REGION Network 9: Clear IDs from HMI if not on that screen
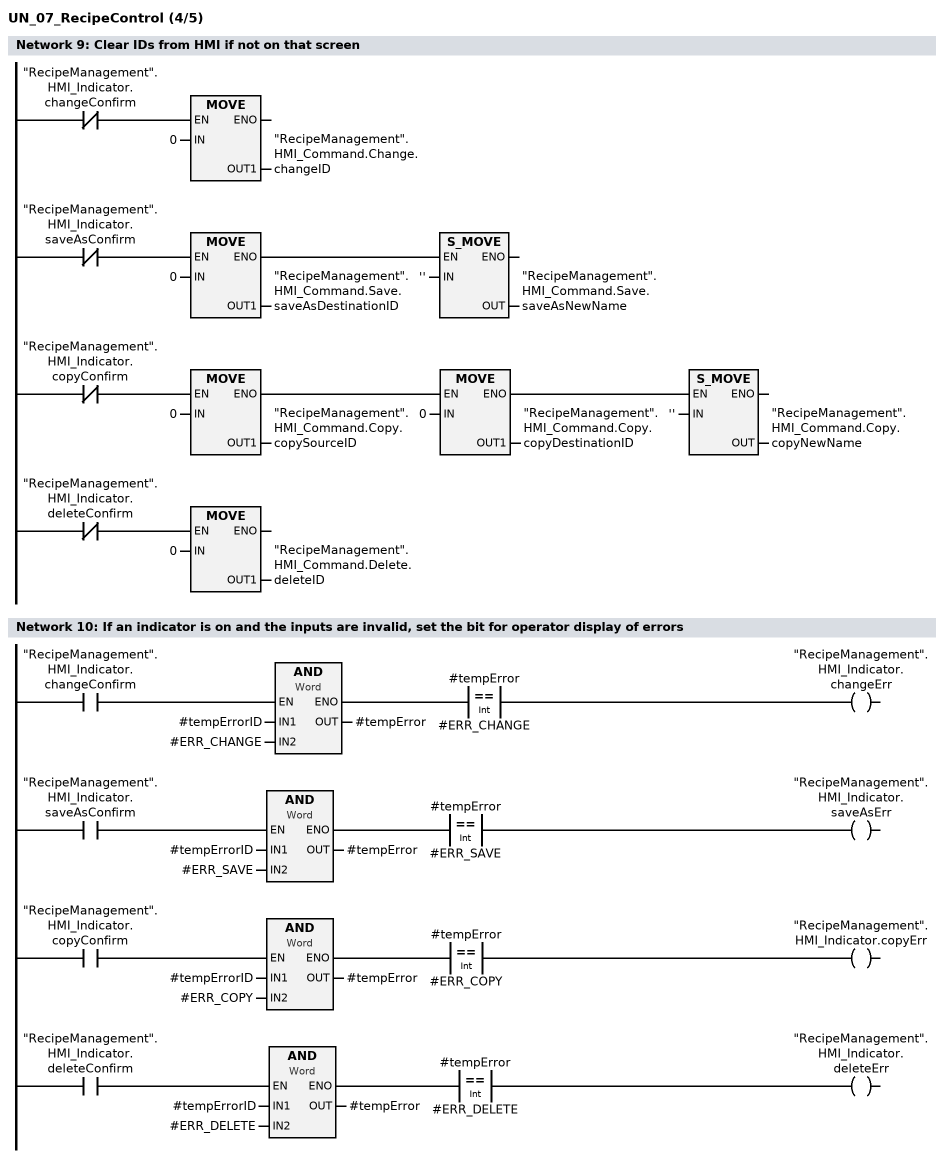
   RUNG wire#powerrail
      I_Contact( "RecipeManagement".HMI_Indicator.changeConfirm )
      Move(in := 0, out1 => "RecipeManagement".HMI_Command.Change.changeID)
   END_RUNG
   RUNG wire#powerrail
      I_Contact( "RecipeManagement".HMI_Indicator.saveAsConfirm )
      Move(in := 0, out1 => "RecipeManagement".HMI_Command.Save.saveAsDestinationID)
      S_Move(in := '', out => "RecipeManagement".HMI_Command.Save.saveAsNewName)
   END_RUNG
   RUNG wire#powerrail
      I_Contact( "RecipeManagement".HMI_Indicator.copyConfirm )
      Move(in := 0, out1 => "RecipeManagement".HMI_Command.Copy.copySourceID)
      Move(in := 0, out1 => "RecipeManagement".HMI_Command.Copy.copyDestinationID)
      S_Move(in := '', out => "RecipeManagement".HMI_Command.Copy.copyNewName)
   END_RUNG
   RUNG wire#powerrail
      I_Contact( "RecipeManagement".HMI_Indicator.deleteConfirm )
      Move(in := 0, out1 => "RecipeManagement".HMI_Command.Delete.deleteID)
   END_RUNG
   // the same network as SCL:
   IF NOT "RecipeManagement".HMI_Indicator.changeConfirm THEN
       "RecipeManagement".HMI_Command.Change.changeID := 0;
   END_IF;
   IF NOT "RecipeManagement".HMI_Indicator.saveAsConfirm THEN
       "RecipeManagement".HMI_Command.Save.saveAsDestinationID := 0;
       "RecipeManagement".HMI_Command.Save.saveAsNewName := '';
   END_IF;
   IF NOT "RecipeManagement".HMI_Indicator.copyConfirm THEN
       "RecipeManagement".HMI_Command.Copy.copySourceID := 0;
       "RecipeManagement".HMI_Command.Copy.copyDestinationID := 0;
       "RecipeManagement".HMI_Command.Copy.copyNewName := '';
   END_IF;
   IF NOT "RecipeManagement".HMI_Indicator.deleteConfirm THEN
       "RecipeManagement".HMI_Command.Delete.deleteID := 0;
   END_IF;
END_REGION

REGION Network 10: If an indicator is on and the inputs are invalid, set the bit for operator display of errors
   RUNG wire#powerrail
      Contact( "RecipeManagement".HMI_Indicator.changeConfirm )
      { S7_Templates := "SrcType := Word" } And(in1 := #tempErrorID, in2 := #ERR_CHANGE, out => #tempError)
      { S7_Templates := "SrcType := Int" } EQ_Contact(in1 := #tempError, in2 := #ERR_CHANGE)
      Coil( "RecipeManagement".HMI_Indicator.changeErr )
   END_RUNG
   RUNG wire#powerrail
      Contact( "RecipeManagement".HMI_Indicator.saveAsConfirm )
      { S7_Templates := "SrcType := Word" } And(in1 := #tempErrorID, in2 := #ERR_SAVE, out => #tempError)
      { S7_Templates := "SrcType := Int" } EQ_Contact(in1 := #tempError, in2 := #ERR_SAVE)
      Coil( "RecipeManagement".HMI_Indicator.saveAsErr )
   END_RUNG
   RUNG wire#powerrail
      Contact( "RecipeManagement".HMI_Indicator.copyConfirm )
      { S7_Templates := "SrcType := Word" } And(in1 := #tempErrorID, in2 := #ERR_COPY, out => #tempError)
      { S7_Templates := "SrcType := Int" } EQ_Contact(in1 := #tempError, in2 := #ERR_COPY)
      Coil( "RecipeManagement".HMI_Indicator.copyErr )
   END_RUNG
   RUNG wire#powerrail
      Contact( "RecipeManagement".HMI_Indicator.deleteConfirm )
      { S7_Templates := "SrcType := Word" } And(in1 := #tempErrorID, in2 := #ERR_DELETE, out => #tempError)
      { S7_Templates := "SrcType := Int" } EQ_Contact(in1 := #tempError, in2 := #ERR_DELETE)
      Coil( "RecipeManagement".HMI_Indicator.deleteErr )
   END_RUNG
   // the same network as SCL:
   IF "RecipeManagement".HMI_Indicator.changeConfirm THEN #tempError := #tempErrorID AND #ERR_CHANGE; END_IF;
   "RecipeManagement".HMI_Indicator.changeErr := "RecipeManagement".HMI_Indicator.changeConfirm AND (#tempError = #ERR_CHANGE);
   IF "RecipeManagement".HMI_Indicator.saveAsConfirm THEN #tempError := #tempErrorID AND #ERR_SAVE; END_IF;
   "RecipeManagement".HMI_Indicator.saveAsErr := "RecipeManagement".HMI_Indicator.saveAsConfirm AND (#tempError = #ERR_SAVE);
   IF "RecipeManagement".HMI_Indicator.copyConfirm THEN #tempError := #tempErrorID AND #ERR_COPY; END_IF;
   "RecipeManagement".HMI_Indicator.copyErr := "RecipeManagement".HMI_Indicator.copyConfirm AND (#tempError = #ERR_COPY);
   IF "RecipeManagement".HMI_Indicator.deleteConfirm THEN #tempError := #tempErrorID AND #ERR_DELETE; END_IF;
   "RecipeManagement".HMI_Indicator.deleteErr := "RecipeManagement".HMI_Indicator.deleteConfirm AND (#tempError = #ERR_DELETE);
END_REGION

REGION Network 11: Call Recipe HMI Manager to handle display of setpoints
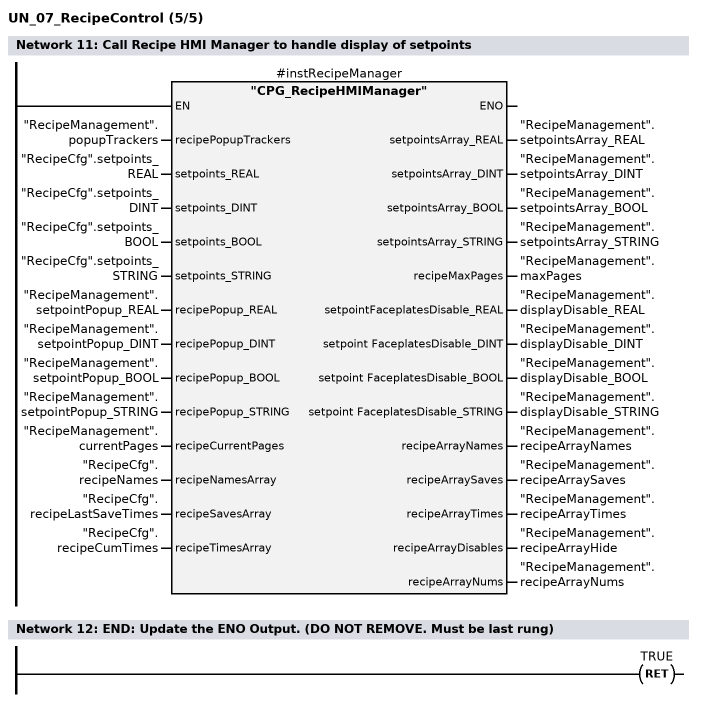
   RUNG wire#powerrail
      #instRecipeManager(recipePopupTrackers := "RecipeManagement".popupTrackers, setpoints_REAL := "RecipeCfg".setpoints_REAL, setpoints_DINT := "RecipeCfg".setpoints_DINT, setpoints_BOOL := "RecipeCfg".setpoints_BOOL, setpoints_STRING := "RecipeCfg".setpoints_STRING, recipePopup_REAL := "RecipeManagement".setpointPopup_REAL, recipePopup_DINT := "RecipeManagement".setpointPopup_DINT, recipePopup_BOOL := "RecipeManagement".setpointPopup_BOOL, recipePopup_STRING := "RecipeManagement".setpointPopup_STRING, recipeCurrentPages := "RecipeManagement".currentPages, recipeNamesArray := "RecipeCfg".recipeNames, recipeSavesArray := "RecipeCfg".recipeLastSaveTimes, recipeTimesArray := "RecipeCfg".recipeCumTimes, setpointsArray_REAL => "RecipeManagement".setpointsArray_REAL, setpointsArray_DINT => "RecipeManagement".setpointsArray_DINT, setpointsArray_BOOL => "RecipeManagement".setpointsArray_BOOL, setpointsArray_STRING => "RecipeManagement".setpointsArray_STRING, recipeMaxPages => "RecipeManagement".maxPages, setpointFaceplatesDisable_REAL => "RecipeManagement".displayDisable_REAL, "setpoint FaceplatesDisable_DINT" => "RecipeManagement".displayDisable_DINT, "setpoint FaceplatesDisable_BOOL" => "RecipeManagement".displayDisable_BOOL, "setpoint FaceplatesDisable_STRING" => "RecipeManagement".displayDisable_STRING, recipeArrayNames => "RecipeManagement".recipeArrayNames, recipeArraySaves => "RecipeManagement".recipeArraySaves, recipeArrayTimes => "RecipeManagement".recipeArrayTimes, recipeArrayDisables => "RecipeManagement".recipeArrayHide, recipeArrayNums => "RecipeManagement".recipeArrayNums)
   END_RUNG
   // the same network as SCL:
   #instRecipeManager(recipePopupTrackers := "RecipeManagement".popupTrackers,   // "CPG_RecipeHMIManager"
                      setpoints_REAL := "RecipeCfg".setpoints_REAL,
                      setpoints_DINT := "RecipeCfg".setpoints_DINT,
                      setpoints_BOOL := "RecipeCfg".setpoints_BOOL,
                      setpoints_STRING := "RecipeCfg".setpoints_STRING,
                      recipePopup_REAL := "RecipeManagement".setpointPopup_REAL,
                      recipePopup_DINT := "RecipeManagement".setpointPopup_DINT,
                      recipePopup_BOOL := "RecipeManagement".setpointPopup_BOOL,
                      recipePopup_STRING := "RecipeManagement".setpointPopup_STRING,
                      recipeCurrentPages := "RecipeManagement".currentPages,
                      recipeNamesArray := "RecipeCfg".recipeNames,
                      recipeSavesArray := "RecipeCfg".recipeLastSaveTimes,
                      recipeTimesArray := "RecipeCfg".recipeCumTimes,
                      setpointsArray_REAL => "RecipeManagement".setpointsArray_REAL,
                      setpointsArray_DINT => "RecipeManagement".setpointsArray_DINT,
                      setpointsArray_BOOL => "RecipeManagement".setpointsArray_BOOL,
                      setpointsArray_STRING => "RecipeManagement".setpointsArray_STRING,
                      recipeMaxPages => "RecipeManagement".maxPages,
                      setpointFaceplatesDisable_REAL => "RecipeManagement".displayDisable_REAL,
                      "setpoint FaceplatesDisable_DINT" => "RecipeManagement".displayDisable_DINT,
                      "setpoint FaceplatesDisable_BOOL" => "RecipeManagement".displayDisable_BOOL,
                      "setpoint FaceplatesDisable_STRING" => "RecipeManagement".displayDisable_STRING,
                      recipeArrayNames => "RecipeManagement".recipeArrayNames,
                      recipeArraySaves => "RecipeManagement".recipeArraySaves,
                      recipeArrayTimes => "RecipeManagement".recipeArrayTimes,
                      recipeArrayDisables => "RecipeManagement".recipeArrayHide,
                      recipeArrayNums => "RecipeManagement".recipeArrayNums);
END_REGION

REGION Network 12: END: Update the ENO Output. (DO NOT REMOVE. Must be last rung)
   RUNG wire#powerrail
      ReturnCoil( TRUE )
   END_RUNG
   // the same network as SCL:
   ENO := TRUE;
   RETURN;
END_REGION
END_FUNCTION_BLOCK

FUNCTION_BLOCK "CPG_RecipeControl"
TITLE = CPG_RecipeControl
{ S7_Optimized_Access := 'TRUE' }
AUTHOR : 'tech.team.motioncontrol@siemens.com'
FAMILY : CPG
VERSION : 1.1
//Support: tech.team.motioncontrol@siemens.com
   VAR_INPUT 
      enable { ExternalAccessible := 'False'; ExternalVisible := 'False'; ExternalWritable := 'False'} : Bool;   // Recipe change is only possible if instruction is enabled
      recipeChangeID { ExternalAccessible := 'False'; ExternalVisible := 'False'; ExternalWritable := 'False'} : Int;   // ID of recipe to change to
      recipeChangeReq { ExternalAccessible := 'False'; ExternalVisible := 'False'; ExternalWritable := 'False'} : Bool;   // Change recipe on rising edge
      recipeSaveReq { ExternalAccessible := 'False'; ExternalVisible := 'False'; ExternalWritable := 'False'} : Bool;   // Save current recipe on rising edge
      recipeSaveAsID { ExternalAccessible := 'False'; ExternalVisible := 'False'; ExternalWritable := 'False'} : Int;   // Location to saveas recipe to
      recipeSaveAsReq { ExternalAccessible := 'False'; ExternalVisible := 'False'; ExternalWritable := 'False'} : Bool;   // SaveAs recipe on rising edge
      recipeCopySourceID { ExternalAccessible := 'False'; ExternalVisible := 'False'; ExternalWritable := 'False'} : Int;   // Location to copy recipe from
      recipeCopyID { ExternalAccessible := 'False'; ExternalVisible := 'False'; ExternalWritable := 'False'} : Int;   // Location to copy recipe to
      recipeCopyReq { ExternalAccessible := 'False'; ExternalVisible := 'False'; ExternalWritable := 'False'} : Bool;   // Copy recipe on rising edge
      newRecipeName { ExternalAccessible := 'False'; ExternalVisible := 'False'; ExternalWritable := 'False'} : String[60];   // Name of the saveas or copied recipe
      recipeDeleteID { ExternalAccessible := 'False'; ExternalVisible := 'False'; ExternalWritable := 'False'} : Int;   // Location of recipe to delete
      recipeDeleteReq { ExternalAccessible := 'False'; ExternalVisible := 'False'; ExternalWritable := 'False'} : Bool;   // Delete recipe on rising edge
      resetAllTimes { ExternalAccessible := 'False'; ExternalVisible := 'False'; ExternalWritable := 'False'} : Bool;   // Reset cumulative seconds for all recipes
   END_VAR

   VAR_OUTPUT 
      currentRecipeID { ExternalAccessible := 'False'; ExternalVisible := 'False'; ExternalWritable := 'False'} : Int;   // ID of the current recipe
      currentRecipeName { ExternalAccessible := 'False'; ExternalVisible := 'False'; ExternalWritable := 'False'} : String[60];   // Name of the current recipe
      recipeChangeDisabled { ExternalAccessible := 'False'; ExternalVisible := 'False'; ExternalWritable := 'False'} : Bool;   // Recipe changes are enabled
      recipeSetpointDiff { ExternalAccessible := 'False'; ExternalVisible := 'False'; ExternalWritable := 'False'} : Bool;   // New setpoint differs from current recipe value
      recipeCurrentSeconds { ExternalAccessible := 'False'; ExternalVisible := 'False'; ExternalWritable := 'False'} : Time;   // Current recipe time in seconds
      error { ExternalAccessible := 'False'; ExternalVisible := 'False'; ExternalWritable := 'False'} : Bool;   // Error Present
      errorID { ExternalAccessible := 'False'; ExternalVisible := 'False'; ExternalWritable := 'False'} : Word := 16#0000;   // Code for Status
   END_VAR

   VAR_IN_OUT 
      recipeControl : "CPG_typeRecipeControl";   // Recipe Control tag
      recipeNames : Array[0.."CPG_NO_OF_RECIPE_UPPER_LIM"] of String[60];   // All recipe names
      recipeCumSeconds : Array[0.."CPG_NO_OF_RECIPE_UPPER_LIM"] of Time;   // Cumulative times for all recipes
      recipeSaveDates {InstructionName := 'DTL'; LibVersion := '1.0'} : Array[0.."CPG_NO_OF_RECIPE_UPPER_LIM"] of DTL;   // Recipe saved date time
   END_VAR

   VAR 
      statSetpoinDiffTimer {InstructionName := 'TON_TIME'; LibVersion := '1.0'; ExternalAccessible := 'False'; ExternalVisible := 'False'; ExternalWritable := 'False'} : TON_TIME;
      statPrevRecipe { ExternalAccessible := 'False'; ExternalVisible := 'False'; ExternalWritable := 'False'} : Int;
      statChangeReq {InstructionName := 'R_TRIG'; LibVersion := '1.0'; ExternalAccessible := 'False'; ExternalVisible := 'False'; ExternalWritable := 'False'} : R_TRIG;
      statSaveReq {InstructionName := 'R_TRIG'; LibVersion := '1.0'; ExternalAccessible := 'False'; ExternalVisible := 'False'; ExternalWritable := 'False'} : R_TRIG;
      statSaveAsReq {InstructionName := 'R_TRIG'; LibVersion := '1.0'; ExternalAccessible := 'False'; ExternalVisible := 'False'; ExternalWritable := 'False'} : R_TRIG;
      statCopyReq {InstructionName := 'R_TRIG'; LibVersion := '1.0'; ExternalAccessible := 'False'; ExternalVisible := 'False'; ExternalWritable := 'False'} : R_TRIG;
      statDeleteReq {InstructionName := 'R_TRIG'; LibVersion := '1.0'; ExternalAccessible := 'False'; ExternalVisible := 'False'; ExternalWritable := 'False'} : R_TRIG;
      statChangeTimer {InstructionName := 'TP_TIME'; LibVersion := '1.0'; ExternalAccessible := 'False'; ExternalVisible := 'False'; ExternalWritable := 'False'} : TP_TIME;
      statChangeTimerFall {InstructionName := 'F_TRIG'; LibVersion := '1.0'; ExternalAccessible := 'False'; ExternalVisible := 'False'; ExternalWritable := 'False'} : F_TRIG;
      statSaveTimer {InstructionName := 'TP_TIME'; LibVersion := '1.0'; ExternalAccessible := 'False'; ExternalVisible := 'False'; ExternalWritable := 'False'} : TP_TIME;
      statSaveTimerFall {InstructionName := 'F_TRIG'; LibVersion := '1.0'; ExternalAccessible := 'False'; ExternalVisible := 'False'; ExternalWritable := 'False'} : F_TRIG;
      statSaveAsTimer {InstructionName := 'TP_TIME'; LibVersion := '1.0'; ExternalAccessible := 'False'; ExternalVisible := 'False'; ExternalWritable := 'False'} : TP_TIME;
      statSaveAsTimerFall {InstructionName := 'F_TRIG'; LibVersion := '1.0'; ExternalAccessible := 'False'; ExternalVisible := 'False'; ExternalWritable := 'False'} : F_TRIG;
      statCopyTimer {InstructionName := 'TP_TIME'; LibVersion := '1.0'; ExternalAccessible := 'False'; ExternalVisible := 'False'; ExternalWritable := 'False'} : TP_TIME;
      statCopyTimerFall {InstructionName := 'F_TRIG'; LibVersion := '1.0'; ExternalAccessible := 'False'; ExternalVisible := 'False'; ExternalWritable := 'False'} : F_TRIG;
      statDeleteTimer {InstructionName := 'TP_TIME'; LibVersion := '1.0'; ExternalAccessible := 'False'; ExternalVisible := 'False'; ExternalWritable := 'False'} : TP_TIME;
      statDeleteTimerFall {InstructionName := 'F_TRIG'; LibVersion := '1.0'; ExternalAccessible := 'False'; ExternalVisible := 'False'; ExternalWritable := 'False'} : F_TRIG;
      statPrevCumSeconds { ExternalAccessible := 'False'; ExternalVisible := 'False'; ExternalWritable := 'False'} : Array[0.."CPG_NO_OF_RECIPE_UPPER_LIM"] of Time;
      statChangeTimeStamp {InstructionName := 'DTL'; LibVersion := '1.0'; ExternalAccessible := 'False'; ExternalVisible := 'False'; ExternalWritable := 'False'} : DTL;
   END_VAR

   VAR_TEMP 
      tempChangeEN : Bool;
      tempCopyRecipeEN : Bool;
      tempSaveRecipeEN : Bool;
      tempDeleteRecipeEN : Bool;
      tempDTLError : Int;
      tempLoop : Int;
      tempTime {InstructionName := 'DTL'; LibVersion := '1.0'} : DTL;
      tempRecipeSaveAs : Bool;
   END_VAR

   VAR CONSTANT 
      MAX_RECIPE_NUM : Int := 20;
      WARNING_TIMERLEN : Time := T#1s;
      CHG_ERR : Word := 16#8001;
      SAVE_ERR : Word := 16#8002;
      COPY_ERR : Word := 16#8004;
      DEL_ERR : Word := 16#8008;
   END_VAR


BEGIN
	//============================================================================================================
	// SIEMENS AG
	// (c)Copyright 2019 All Rights Reserved
	//------------------------------------------------------------------------------------------------------------
	// Library: LCPG
	// Tested with: S7-1500 with FW version V2.1
	// Engineering: TIA Portal V14
	// Restrictions: ---
	// Requirements: S7-1500
	// Functionality: used to control the current machine recipe
	// Support: tech.team.motioncontrol@siemens.com
	//------------------------------------------------------------------------------------------------------------
	// Change log table:
	// Version       Date               Expert in charge    Changes applied
	//  01.01.00     02.01.2019         KB                  Initial Release
	//============================================================================================================
	// Function : CPG_RecipeControl
	//============================================================================================================
	
	REGION INITIALIZATION
	    #errorID := 16#0000;
	    
	    #recipeControl.RecipeChangeDisabled := NOT #enable;
	    
	    //check lanugage for out of bounds
	    IF (#recipeControl.LanguageSelection < 0) OR (#recipeControl.LanguageSelection > "LPMLV30_LANGUAGES_UPPER_LIM") THEN
	        #errorID := #errorID OR 16#1000;
	        #recipeControl.LanguageSelection := 0;
	    END_IF;
	    
	    
	    //Dectect any recipe & setpoint differences
	    //if any call of recipe setpoint FBs has a difference, the RecipeSetpointDiff bit is set
	    IF #recipeControl.RecipeSetpointDiff THEN
	        #recipeSetpointDiff := true;
	        #recipeControl.RecipeSetpointDiff := false;
	    END_IF;
	END_REGION
	
	
	REGION RECIPE MANAGEMENT ENABLING
	    //Check that only 1 recipe command is active
	    IF NOT (#recipeControl.RecipeCopy OR #recipeControl.RecipeDelete OR #recipeControl.RecipeSave) THEN     //all false except change
	        #tempChangeEN := true;
	    END_IF;
	    IF NOT (#recipeControl.RecipeCopy OR #recipeControl.RecipeDelete OR #recipeControl.RecipeChange) THEN   //all false except save/saveas
	        #tempSaveRecipeEN := true;
	    END_IF;
	    IF NOT (#recipeControl.RecipeChange OR #recipeControl.RecipeDelete OR #recipeControl.RecipeSave) THEN   //all false except copy
	        #tempCopyRecipeEN := true;
	    END_IF;
	    IF NOT (#recipeControl.RecipeCopy OR #recipeControl.RecipeChange OR #recipeControl.RecipeSave) THEN     //all false except delete
	        #tempDeleteRecipeEN := true;
	    END_IF;
	    
	    
	    //RecipeCmd out of bounds, or equal to the current recipe
	    IF (#recipeChangeID > #MAX_RECIPE_NUM) OR (#recipeChangeID < 0) OR (#recipeChangeID = #recipeControl.CurrentRecipeID) THEN
	        #errorID := #errorID OR #CHG_ERR;
	        #tempChangeEN := false;
	    END_IF;
	    //RecipeSaveAsCmd out of bounds, or attempting to over current recipe
	    IF (#recipeSaveAsID > #MAX_RECIPE_NUM) OR (#recipeSaveAsID < 0) OR (#recipeSaveAsID = #recipeControl.CurrentRecipeID) THEN
	        #errorID := #errorID OR #SAVE_ERR;
	        #tempSaveRecipeEN := false;
	    END_IF;
	    //RecipeCopyCmd or RecipeCopySourceCmd out of bounds, cannot copy to currently running recipe
	    IF (#recipeCopyID > #MAX_RECIPE_NUM) OR (#recipeCopyID < 0) OR (#recipeCopySourceID > #MAX_RECIPE_NUM) OR (#recipeCopySourceID < 0)
	        OR #recipeCopyID = #recipeControl.CurrentRecipeID THEN
	        #errorID := #errorID OR #COPY_ERR;
	        #tempCopyRecipeEN := false;
	    END_IF;
	    //RecipeDeleteCmd out of bounds or equal to current recipe
	    IF (#recipeDeleteID > #MAX_RECIPE_NUM) OR (#recipeDeleteID < 0) OR (#recipeDeleteID = #recipeControl.CurrentRecipeID) THEN
	        #errorID := #errorID OR #DEL_ERR;
	        #tempDeleteRecipeEN := false;
	    END_IF;
	END_REGION
	
	
	REGION RECIPE CHANGE
	    //only allow recipe changes while enabled
	    IF #enable THEN
	        
	        //timer needed for display & troubleshooting
	        //timer starts on rising edge of the req signal and persists for 1s
	        #statChangeReq(CLK := #recipeChangeReq);
	        
	        #statChangeTimer(IN := #statChangeReq.Q,
	                     PT := #WARNING_TIMERLEN);
	        
	        #statChangeTimerFall(CLK := #statChangeTimer.Q);
	        
	        
	        //Check that the recipe to change is valid & no other command is active
	        IF #tempChangeEN THEN
	            
	            //set output to indicate that a recipe is being changed
	            IF #statChangeTimer.Q THEN
	                #recipeControl.RecipeChange := true;
	            ELSE
	                #recipeControl.RecipeChange := false;
	            END_IF;
	            
	            //change recipe on done bit, true for only 1 scan
	            IF #statChangeTimerFall.Q THEN
	                #recipeControl.RecipeChangeNum := #recipeControl.RecipeChangeNum + 1;
	                #recipeControl.CurrentRecipeID := #recipeChangeID;
	                #recipeControl.CurrentRecipeName := #recipeNames[#recipeControl.CurrentRecipeID];
	            END_IF;
	            
	        END_IF;
	        
	    END_IF;
	END_REGION
	
	
	REGION RECIPE SAVEAS
	    //timer needed for display & troubleshooting
	    //timer starts on rising edge of the req signal and persists for 1s
	    #statSaveAsReq(CLK := #recipeSaveAsReq);
	    
	    #statSaveAsTimer(IN := #statSaveAsReq.Q,
	                 PT := #WARNING_TIMERLEN);
	    
	    #statSaveAsTimerFall(CLK := #statSaveAsTimer.Q);
	    
	    
	    //Check that the recipe to save is valid & no other command is active
	    IF #tempSaveRecipeEN THEN
	        
	        //set output to indicate that a recipe is being saved
	        //because Save & SaveAs use the same output (RecipeControl.RecipeSave), this is handled slightly differently
	        IF #statSaveAsTimer.Q THEN
	            #tempRecipeSaveAs := true;
	        END_IF;
	        
	        
	        //set work variables so that setpoints know the source/destination of the copy operation
	        IF #statSaveAsTimer.Q THEN
	            #recipeControl.RecipeSourceID := #recipeControl.CurrentRecipeID;
	            #recipeControl.RecipeDestinationID := #recipeSaveAsID;
	        END_IF;
	        
	        //update counter, take timestamp, and update recipe name
	        IF #statSaveAsTimerFall.Q THEN
	            #recipeControl.RecipeSaveNum := #recipeControl.RecipeSaveNum + 1;
	            #tempDTLError := RD_LOC_T(#recipeSaveDates[#recipeControl.RecipeDestinationID]);
	            #recipeNames[#recipeControl.RecipeDestinationID] := #newRecipeName;
	        END_IF;
	        
	    END_IF;
	END_REGION
	
	
	REGION RECIPE SAVE
	    //timer needed for display & troubleshooting
	    //timer starts on rising edge of the req signal and persists for 1s
	    #statSaveReq(CLK := #recipeSaveReq);
	    
	    #statSaveTimer(IN := #statSaveReq.Q,
	               PT := #WARNING_TIMERLEN);
	    
	    #statSaveTimerFall(CLK := #statSaveTimer.Q);
	    
	    
	    //saving is always possible
	    //note that the saveas REGION must be after the save REGION
	    //otherwise RecipeControl.RecipeSave won't be set by a saveas
	    
	    //set output to indicate that a recipe is being saved
	    //because Save & SaveAs use the same output (RecipeControl.RecipeSave), this is handled slightly differently
	    IF #statSaveTimer.Q  OR #tempRecipeSaveAs THEN
	        #recipeControl.RecipeSave := true;
	    ELSE
	        #recipeControl.RecipeSave := false;
	    END_IF;
	    
	    //set work variables so that setpoints know the source/destination of the save operation
	    IF #statSaveTimer.Q THEN
	        #recipeControl.RecipeSourceID := #recipeControl.CurrentRecipeID;
	        #recipeControl.RecipeDestinationID := #recipeControl.CurrentRecipeID;
	    END_IF;
	    
	    //update counter, take timestamp
	    IF #statSaveTimerFall.Q THEN
	        #recipeControl.RecipeSaveNum := #recipeControl.RecipeSaveNum + 1;
	        #tempDTLError := RD_LOC_T(#recipeSaveDates[#recipeControl.RecipeDestinationID]);
	    END_IF;
	END_REGION
	
	
	REGION RECIPE COPY
	    //timer needed for display & troubleshooting
	    //timer starts on rising edge of the req signal and persists for 1s
	    #statCopyReq(CLK := #recipeCopyReq);
	    
	    #statCopyTimer(IN := #statCopyReq.Q,
	               PT := #WARNING_TIMERLEN);
	    
	    #statCopyTimerFall(CLK := #statCopyTimer.Q);
	    
	    
	    //Check that the recipes to copy are valid & no other command is active
	    IF #tempCopyRecipeEN THEN
	        
	        //set output to indicate that a recipe is being copied
	        IF #statCopyTimer.Q THEN
	            #recipeControl.RecipeCopy := true;
	        ELSE
	            #recipeControl.RecipeCopy := false;
	        END_IF;
	        
	        //set work variables so that setpoints know the source/destination of the copy operation
	        IF #statCopyTimer.Q THEN
	            #recipeControl.RecipeSourceID := #recipeCopySourceID;
	            #recipeControl.RecipeDestinationID := #recipeCopyID;
	        END_IF;
	        
	        //update the recipename of the new recipe, increment change work variable
	        IF #statCopyTimerFall.Q THEN
	            #recipeControl.RecipeCopyNum := #recipeControl.RecipeCopyNum + 1;
	            #tempDTLError := RD_LOC_T(#recipeSaveDates[#recipeControl.RecipeDestinationID]);
	            #recipeNames[#recipeControl.RecipeDestinationID] := #newRecipeName;
	        END_IF;
	        
	    END_IF;
	END_REGION
	
	
	REGION RECIPE DELETE
	    //timer needed for display & troubleshooting
	    //timer starts on rising edge of the req signal and persists for 1s
	    #statDeleteReq(CLK := #recipeDeleteReq);
	    
	    #statDeleteTimer(IN := #statDeleteReq.Q,
	                 PT := #WARNING_TIMERLEN);
	    
	    #statDeleteTimerFall(CLK := #statDeleteTimer.Q);
	    
	    
	    //Check that the recipe to delete is valid & no other command is active
	    IF #tempDeleteRecipeEN THEN
	        
	        //set output to indicate that a recipe is being copied
	        IF #statDeleteTimer.Q THEN
	            #recipeControl.RecipeDelete := true;
	        ELSE
	            #recipeControl.RecipeDelete := false;
	        END_IF;
	        
	        //set work variable so that setpoints know the destination of the delete operation
	        IF #statDeleteTimer.Q THEN
	            #recipeControl.RecipeDestinationID := #recipeDeleteID;
	        END_IF;
	        
	        //clear the recipe name
	        IF #statDeleteTimerFall.Q THEN
	            #recipeControl.RecipeDeleteNum := #recipeControl.RecipeDeleteNum + 1;
	            #tempDTLError := RD_LOC_T(#recipeSaveDates[#recipeControl.RecipeDestinationID]);
	            #recipeNames[#recipeControl.RecipeDestinationID] := '';
	        END_IF;
	        
	    END_IF;
	END_REGION
	
	
	REGION TIME TRACKING
	    //reset all times resets the cumulative time for all recipes, and the cum seconds output, but does not change the save timestamps
	    IF #resetAllTimes THEN
	        FOR #tempLoop := 0 TO #MAX_RECIPE_NUM DO
	            // set all cumulative times to zero
	            #recipeCumSeconds[#tempLoop] := T#0s;
	            #statPrevCumSeconds[#tempLoop] := T#0s;
	        END_FOR;
	        #recipeCurrentSeconds := T#0s;
	    END_IF;
	    
	    //if recipe changes, note the time of change and save the accumulated time for the 
	    IF #recipeControl.CurrentRecipeID <> #statPrevRecipe THEN
	        #tempDTLError := RD_LOC_T(#statChangeTimeStamp);
	        #statPrevCumSeconds[#recipeControl.CurrentRecipeID] := #recipeCumSeconds[#recipeControl.CurrentRecipeID];
	        #recipeCurrentSeconds := T#0s;
	    END_IF;
	    
	    //must initialize this value or timetracking does not work on plc startup
	    IF #statChangeTimeStamp = DTL#1970-01-01-00:00:00 THEN
	        #tempDTLError := RD_LOC_T(#statChangeTimeStamp);
	    END_IF;
	    
	    #tempDTLError := RD_LOC_T(#tempTime);
	    #recipeCurrentSeconds := T_DIFF(IN1 := #tempTime, IN2 := #statChangeTimeStamp);
	    #recipeCumSeconds[#recipeControl.CurrentRecipeID] := #statPrevCumSeconds[#recipeControl.CurrentRecipeID] + #recipeCurrentSeconds;
	END_REGION
	
	
	REGION SET OUTPUTS
	    //Update current recipe name in case user changed RecipeControl.CurrentRecipeName on the HMI
	    IF #recipeControl.CurrentRecipeName <> #recipeNames[#recipeControl.CurrentRecipeID] THEN
	        #recipeNames[#recipeControl.CurrentRecipeID] := #recipeControl.CurrentRecipeName;
	    ELSE
	        #recipeControl.CurrentRecipeName := #recipeNames[#recipeControl.CurrentRecipeID];
	    END_IF;
	    
	    //tmpDTLerror recieves a value if there is an eror returning the PLC system time
	    IF #tempDTLError <> 0 THEN
	        #errorID := #errorID OR 16#0100;
	    END_IF;
	    
	    //report error bit
	    IF #errorID = 16#0 THEN
	        #error := false;
	    ELSE
	        #error := true;
	    END_IF;
	    
	    //ensure recipe display numbers are in bounds
	    #recipeControl.RecipeID_A := LIMIT(MN := 0, IN := #recipeControl.RecipeID_A, MX := #MAX_RECIPE_NUM);
	    #recipeControl.RecipeID_B := LIMIT(MN := 0, IN := #recipeControl.RecipeID_B, MX := #MAX_RECIPE_NUM);
	    #recipeControl.RecipeID_C := LIMIT(MN := 0, IN := #recipeControl.RecipeID_C, MX := #MAX_RECIPE_NUM);
	    
	    //set some final outputs
	    #statPrevRecipe := #recipeControl.CurrentRecipeID;
	    #currentRecipeID := #recipeControl.CurrentRecipeID;
	    #currentRecipeName := #recipeControl.CurrentRecipeName;
	    #recipeChangeDisabled := #recipeControl.RecipeChangeDisabled;
	END_REGION
	
	//  -------------- END OF LOGIC -------------------------
	ENO := TRUE;   // Set the ENO output
END_FUNCTION_BLOCK

FUNCTION_BLOCK "CPG_RecipeHMIManager"
TITLE = CPG_RecipeHMIManager
{ S7_Optimized_Access := 'TRUE' }
AUTHOR : 'tech.team.motioncontrol@siemens.com'
FAMILY : CPG
VERSION : 1.1
//Support: tech.team.motioncontrol@siemens.com
   VAR_INPUT 
      recipePopupTrackers { ExternalAccessible := 'False'; ExternalVisible := 'False'; ExternalWritable := 'False'} : Array[0..#NUM_TYPES] of Int;   // Index of recipe that is to be displayed in popup
   END_VAR

   VAR_OUTPUT 
      setpointsArray_REAL { ExternalAccessible := 'False'; ExternalVisible := 'False'; ExternalWritable := 'False'} : Array[0..11] of "CPG_typeRecipeSetpoint_REAL";   // Setpoints to display
      setpointsArray_DINT { ExternalAccessible := 'False'; ExternalVisible := 'False'; ExternalWritable := 'False'} : Array[0..11] of "CPG_typeRecipeSetpoint_DINT";   // Setpoints to display
      setpointsArray_BOOL { ExternalAccessible := 'False'; ExternalVisible := 'False'; ExternalWritable := 'False'} : Array[0..11] of "CPG_typeRecipeSetpoint_BOOL";   // Setpoints to display
      setpointsArray_STRING { ExternalAccessible := 'False'; ExternalVisible := 'False'; ExternalWritable := 'False'} : Array[0..11] of "CPG_typeRecipeSetpoint_STRING";   // Setpoints to display
      recipeMaxPages { ExternalAccessible := 'False'; ExternalVisible := 'False'; ExternalWritable := 'False'} : Array[0..4] of Int;   // Max pages for all types of setpoint
      setpointFaceplatesDisable_REAL { ExternalAccessible := 'False'; ExternalVisible := 'False'; ExternalWritable := 'False'} : Array[0..11] of Bool;   // True if that setpoint should be hidden
      "setpoint FaceplatesDisable_DINT" { ExternalAccessible := 'False'; ExternalVisible := 'False'; ExternalWritable := 'False'} : Array[0..11] of Bool;   // True if that setpoint should be hidden
      "setpoint FaceplatesDisable_BOOL" { ExternalAccessible := 'False'; ExternalVisible := 'False'; ExternalWritable := 'False'} : Array[0..11] of Bool;   // True if that setpoint should be hidden
      "setpoint FaceplatesDisable_STRING" { ExternalAccessible := 'False'; ExternalVisible := 'False'; ExternalWritable := 'False'} : Array[0..11] of Bool;   // True if that setpoint should be hidden
      recipeArrayNames { ExternalAccessible := 'False'; ExternalVisible := 'False'; ExternalWritable := 'False'} : Array[0..19] of String[60];   // Recipe names to display
      recipeArraySaves {InstructionName := 'DTL'; LibVersion := '1.0'; ExternalAccessible := 'False'; ExternalVisible := 'False'; ExternalWritable := 'False'} : Array[0..19] of DTL;   // Recipe save times to display
      recipeArrayTimes { ExternalAccessible := 'False'; ExternalVisible := 'False'; ExternalWritable := 'False'} : Array[0..19] of Time;   // Recipe cumtimes to display
      recipeArrayDisables { ExternalAccessible := 'False'; ExternalVisible := 'False'; ExternalWritable := 'False'} : Array[0..19] of Bool;   // True if that recipe should be hidden
      recipeArrayNums { ExternalAccessible := 'False'; ExternalVisible := 'False'; ExternalWritable := 'False'} : Array[0..19] of Int;   // Recipe numbers to display
   END_VAR

   VAR_IN_OUT 
      setpoints_REAL : Array[*] of "CPG_typeRecipeSetpoint_REAL";   // Machine setpoints
      setpoints_DINT : Array[*] of "CPG_typeRecipeSetpoint_DINT";   // Machine setpoints
      setpoints_BOOL : Array[*] of "CPG_typeRecipeSetpoint_BOOL";   // Machine setpoints
      setpoints_STRING : Array[*] of "CPG_typeRecipeSetpoint_STRING";   // Machine setpoints
      recipePopup_REAL : "CPG_typeRecipeSetpoint_REAL";   // Tag of popup
      recipePopup_DINT : "CPG_typeRecipeSetpoint_DINT";   // Tag of popup
      recipePopup_BOOL : "CPG_typeRecipeSetpoint_BOOL";   // Tag of popup
      recipePopup_STRING : "CPG_typeRecipeSetpoint_STRING";   // Tag of popup
      recipeCurrentPages : Array[0..4] of Int;   // Current page for viewing setpoints/recipies
      recipeNamesArray : Array[*] of String[60];   // Recipe names
      recipeSavesArray {InstructionName := 'DTL'; LibVersion := '1.0'} : Array[*] of DTL;   // Recipe saves
      recipeTimesArray : Array[*] of Time;   // Recipe cumtimes
   END_VAR

   VAR 
      statPrevCurrentPages { ExternalAccessible := 'False'; ExternalVisible := 'False'; ExternalWritable := 'False'} : Array[0..4] of Int := [4(-1)];
      statPrevPopupTrackers { ExternalAccessible := 'False'; ExternalVisible := 'False'; ExternalWritable := 'False'} : Array[0..#NUM_TYPES] of Int := [4(-1)];
      statPrevPopupsSave { ExternalAccessible := 'False'; ExternalVisible := 'False'; ExternalWritable := 'False'} : Array[0..#NUM_TYPES] of Bool;
      statPrevPopupsRevert { ExternalAccessible := 'False'; ExternalVisible := 'False'; ExternalWritable := 'False'} : Array[0..#NUM_TYPES] of Bool;
      statPrevPopupIN_REAL { ExternalAccessible := 'False'; ExternalVisible := 'False'; ExternalWritable := 'False'} : Real;
      statPrevSetpointIN_REAL { ExternalAccessible := 'False'; ExternalVisible := 'False'; ExternalWritable := 'False'} : Real;
      statPrevPopupIN_DINT { ExternalAccessible := 'False'; ExternalVisible := 'False'; ExternalWritable := 'False'} : DInt;
      statPrevSetpointIN_DINT { ExternalAccessible := 'False'; ExternalVisible := 'False'; ExternalWritable := 'False'} : DInt;
      statPrevPopupIn_BOOL { ExternalAccessible := 'False'; ExternalVisible := 'False'; ExternalWritable := 'False'} : Bool;
      statPrevSetpointIn_BOOL { ExternalAccessible := 'False'; ExternalVisible := 'False'; ExternalWritable := 'False'} : Bool;
      statPrevPopupIn_STRING { ExternalAccessible := 'False'; ExternalVisible := 'False'; ExternalWritable := 'False'} : String[60];
      statPrevSetpointIn_STRING { ExternalAccessible := 'False'; ExternalVisible := 'False'; ExternalWritable := 'False'} : String[60];
   END_VAR

   VAR_TEMP 
      tempLoop : Int;
      tempSetptsLower : Array[0..#NUM_TYPES] of Int;
      tempSetptsUpper : Array[0..#NUM_TYPES] of Int;
      tempCurrentPopup : Int;
      tempNumRecipesLower : Int;
      tempNumRecipesUpper : Int;
   END_VAR

   VAR CONSTANT 
      NUM_TYPES : Int := 3;
      SETPOINTS_PERPAGE : Int := 12;
      RECIPES_PERPAGE : Int := 20;
      INDEX_REAL : Int := 0;
      INDEX_DINT : Int := 1;
      INDEX_BOOL : Int := 2;
      INDEX_STRING : Int := 3;
   END_VAR


BEGIN
	//============================================================================================================
	// SIEMENS AG
	// (c)Copyright 2019 All Rights Reserved
	//------------------------------------------------------------------------------------------------------------
	// Library: LCPG
	// Tested with: S7-1500 with FW version V2.1
	// Engineering: TIA Portal V14
	// Restrictions: ---
	// Requirements: S7-1500
	// Functionality: handles the automatic display of setpoints/recipies
	// Support: tech.team.motioncontrol@siemens.com
	//------------------------------------------------------------------------------------------------------------
	// Change log table:
	// Version       Date               Expert in charge    Changes applied
	//  01.01.00     02.01.2019         KB                  Initial Release
	//============================================================================================================
	// Function : CPG_RecipeHMIManager
	//============================================================================================================
	//
	
	//This function handles the automatic display of the four types of setpoints and the list of recipies
	//There can be any number of setpoints or recipies, but only 12 setpoints and 20 recipies will fit on the screen
	//This block copies 12 of the setpoints into an auxillary array, which is actually displayed on the screen
	//Which 12 setpoints are copied depends on the current page
	//A similar procedure is carried out for the 20 recipe names displayed on the "Recipe_Control" screen
	//Lastly, the recipe that's currently selected is loaded into the popup tag,
	//and any changes made to that tag are propogated back into the "true" setpoint tag
	//The user generally will not need to modify the contents of this block
	
	
	REGION CALCULATE BOUNDS
	    //calculate upper and lower limits 
	    #tempSetptsLower[0] := DINT_TO_INT(LOWER_BOUND(ARR := #setpoints_REAL, DIM := 1));
	    #tempSetptsLower[1] := DINT_TO_INT(LOWER_BOUND(ARR := #setpoints_DINT, DIM := 1));
	    #tempSetptsLower[2] := DINT_TO_INT(LOWER_BOUND(ARR := #setpoints_BOOL, DIM := 1));
	    #tempSetptsLower[3] := DINT_TO_INT(LOWER_BOUND(ARR := #setpoints_STRING, DIM := 1));
	    #tempNumRecipesLower := DINT_TO_INT(LOWER_BOUND(ARR := #recipeNamesArray, DIM := 1));
	    
	    #tempSetptsUpper[0] := DINT_TO_INT(UPPER_BOUND(ARR := #setpoints_REAL, DIM := 1));
	    #tempSetptsUpper[1] := DINT_TO_INT(UPPER_BOUND(ARR := #setpoints_DINT, DIM := 1));
	    #tempSetptsUpper[2] := DINT_TO_INT(UPPER_BOUND(ARR := #setpoints_BOOL, DIM := 1));
	    #tempSetptsUpper[3] := DINT_TO_INT(UPPER_BOUND(ARR := #setpoints_STRING, DIM := 1));
	    #tempNumRecipesUpper := DINT_TO_INT(UPPER_BOUND(ARR := #recipeNamesArray, DIM := 1));
	    
	    FOR #tempLoop := 0 TO #NUM_TYPES DO
	        //calculate max # of pages
	        #recipeMaxPages[#tempLoop] := DINT_TO_INT(CEIL((#tempSetptsUpper[#tempLoop] - #tempSetptsLower[#tempLoop] + 1.0) / #SETPOINTS_PERPAGE));
	        //ensure that current page is within the limits
	        #recipeCurrentPages[#tempLoop] := LIMIT(MN := 1, IN := #recipeCurrentPages[#tempLoop], MX := #recipeMaxPages[#tempLoop]);
	    END_FOR;
	    
	    #recipeMaxPages[4] := DINT_TO_INT(CEIL((#tempNumRecipesUpper - #tempNumRecipesLower + 1.0) / #RECIPES_PERPAGE));
	    #recipeCurrentPages[4] := LIMIT(MN := 1, IN := #recipeCurrentPages[4], MX := #recipeMaxPages[4]);
	END_REGION
	
	
	REGION REAL
	    //index in Setpoints_XXX of the current popup
	    #tempCurrentPopup := #recipePopupTrackers[#INDEX_REAL] + #SETPOINTS_PERPAGE * (#recipeCurrentPages[#INDEX_REAL] - 1) + #tempSetptsLower[#INDEX_REAL];
	    
	    IF #statPrevPopupTrackers[#INDEX_REAL] <> #recipePopupTrackers[#INDEX_REAL] THEN
	        //if a new popup has been loaded, load the new setpoint so they can be displayed
	        #recipePopup_REAL := #setpoints_REAL[#tempCurrentPopup];
	    ELSE
	        //if the HMI popup was updated, relay the commands back to the actual setpoint tag for processing
	        //taking care to ensure that changes to the setpoints tags made in other areas of the program do not get overwritten
	        IF (#statPrevPopupIN_REAL <> #recipePopup_REAL.IN) AND (#statPrevSetpointIN_REAL = #setpoints_REAL[#tempCurrentPopup].IN) THEN
	            #setpoints_REAL[#tempCurrentPopup].IN := #recipePopup_REAL.IN;
	        END_IF;
	        IF #statPrevPopupsSave[#INDEX_REAL] <> #recipePopup_REAL.SaveSetpoint THEN
	            #setpoints_REAL[#tempCurrentPopup].SaveSetpoint := #recipePopup_REAL.SaveSetpoint;
	        END_IF;
	        IF #statPrevPopupsRevert[#INDEX_REAL] <> #recipePopup_REAL.RevertSetpoint THEN
	            #setpoints_REAL[#tempCurrentPopup].RevertSetpoint := #recipePopup_REAL.RevertSetpoint;
	        END_IF;
	        
	        //then update the popup with the latest setpoint information
	        #recipePopup_REAL := #setpoints_REAL[#tempCurrentPopup];
	    END_IF;
	    
	    //set previous values for next scan
	    #statPrevPopupIN_REAL := #recipePopup_REAL.IN;
	    #statPrevSetpointIN_REAL := #setpoints_REAL[#tempCurrentPopup].IN;
	    #statPrevPopupsSave[#INDEX_REAL] := #recipePopup_REAL.SaveSetpoint;
	    #statPrevPopupsRevert[#INDEX_REAL] := #recipePopup_REAL.RevertSetpoint;
	    
	    
	    //update main setpoint display with setpoint data
	    FOR #tempLoop := 0 TO #SETPOINTS_PERPAGE - 1 DO
	        IF #tempLoop + #SETPOINTS_PERPAGE * (#recipeCurrentPages[#INDEX_REAL] - 1) + #tempSetptsLower[#INDEX_REAL] <= #tempSetptsUpper[#INDEX_REAL] THEN
	            #setpointsArray_REAL[#tempLoop] := #setpoints_REAL[#tempLoop + #SETPOINTS_PERPAGE * (#recipeCurrentPages[#INDEX_REAL] - 1) + #tempSetptsLower[#INDEX_REAL]];
	            #setpointFaceplatesDisable_REAL[#tempLoop] := false;
	        ELSE
	            #setpointFaceplatesDisable_REAL[#tempLoop] := true;
	        END_IF;
	    END_FOR;
	END_REGION
	
	
	REGION DINT
	    //index in Setpoints_XXX of the current popup
	    #tempCurrentPopup := #recipePopupTrackers[#INDEX_DINT] + #SETPOINTS_PERPAGE * (#recipeCurrentPages[#INDEX_DINT] - 1) + #tempSetptsLower[#INDEX_DINT];
	    
	    IF #statPrevPopupTrackers[#INDEX_DINT] <> #recipePopupTrackers[#INDEX_DINT] THEN
	        //if a new popup has been loaded, load the new setpoint so they can be displayed
	        #recipePopup_DINT := #setpoints_DINT[#tempCurrentPopup];
	    ELSE
	        //if the HMI popup was updated, relay the commands back to the actual setpoint tag for processing
	        //taking care to ensure that changes to the setpoints tags made in other areas of the program do not get overwritten
	        IF (#statPrevPopupIN_DINT <> #recipePopup_DINT.IN) AND (#statPrevSetpointIN_DINT = #setpoints_DINT[#tempCurrentPopup].IN) THEN
	            #setpoints_DINT[#tempCurrentPopup].IN := #recipePopup_DINT.IN;
	        END_IF;
	        IF #statPrevPopupsSave[#INDEX_DINT] <> #recipePopup_DINT.SaveSetpoint THEN
	            #setpoints_DINT[#tempCurrentPopup].SaveSetpoint := #recipePopup_DINT.SaveSetpoint;
	        END_IF;
	        IF #statPrevPopupsRevert[#INDEX_DINT] <> #recipePopup_DINT.RevertSetpoint THEN
	            #setpoints_DINT[#tempCurrentPopup].RevertSetpoint := #recipePopup_DINT.RevertSetpoint;
	        END_IF;
	        
	        //then update the popup with the latest setpoint information
	        #recipePopup_DINT := #setpoints_DINT[#tempCurrentPopup];
	    END_IF;
	    
	    //set previous values for next scan
	    #statPrevPopupIN_DINT := #recipePopup_DINT.IN;
	    #statPrevSetpointIN_DINT := #setpoints_DINT[#tempCurrentPopup].IN;
	    #statPrevPopupsSave[#INDEX_DINT] := #recipePopup_DINT.SaveSetpoint;
	    #statPrevPopupsRevert[#INDEX_DINT] := #recipePopup_DINT.RevertSetpoint;
	    
	    
	    //update main setpoint display with setpoint data
	    FOR #tempLoop :=  0 TO #SETPOINTS_PERPAGE - 1 DO
	        IF #tempLoop + #SETPOINTS_PERPAGE * (#recipeCurrentPages[#INDEX_DINT] - 1) + #tempSetptsLower[#INDEX_DINT] <= #tempSetptsUpper[#INDEX_DINT] THEN
	            #setpointsArray_DINT[#tempLoop] := #setpoints_DINT[#tempLoop + #SETPOINTS_PERPAGE * (#recipeCurrentPages[#INDEX_DINT] - 1) + #tempSetptsLower[#INDEX_DINT]];
	            #"setpoint FaceplatesDisable_DINT"[#tempLoop] := false;
	        ELSE
	            #"setpoint FaceplatesDisable_DINT"[#tempLoop] := true;
	        END_IF;
	    END_FOR;
	END_REGION
	
	
	REGION BOOL
	    //index in Setpoints_XXX of the current popup
	    #tempCurrentPopup := #recipePopupTrackers[#INDEX_BOOL] + #SETPOINTS_PERPAGE * (#recipeCurrentPages[#INDEX_BOOL] - 1) + #tempSetptsLower[#INDEX_BOOL];
	    
	    IF #statPrevPopupTrackers[#INDEX_BOOL] <> #recipePopupTrackers[#INDEX_BOOL] THEN
	        //if a new popup has been loaded, load the new setpoint so they can be displayed
	        #recipePopup_BOOL := #setpoints_BOOL[#tempCurrentPopup];
	    ELSE
	        //if the HMI popup was updated, relay the commands back to the actual setpoint tag for processing
	        //taking care to ensure that changes to the setpoints tags made in other areas of the program do not get overwritten
	        IF (#statPrevPopupIn_BOOL <> #recipePopup_BOOL.IN) AND (#statPrevSetpointIn_BOOL = #setpoints_BOOL[#tempCurrentPopup].IN) THEN
	            #setpoints_BOOL[#tempCurrentPopup].IN := #recipePopup_BOOL.IN;
	        END_IF;
	        IF #statPrevPopupsSave[#INDEX_BOOL] <> #recipePopup_BOOL.SaveSetpoint THEN
	            #setpoints_BOOL[#tempCurrentPopup].SaveSetpoint := #recipePopup_BOOL.SaveSetpoint;
	        END_IF;
	        IF #statPrevPopupsRevert[#INDEX_BOOL] <> #recipePopup_BOOL.RevertSetpoint THEN
	            #setpoints_BOOL[#tempCurrentPopup].RevertSetpoint := #recipePopup_BOOL.RevertSetpoint;
	        END_IF;
	        
	        //then update the popup with the latest setpoint information
	        #recipePopup_BOOL := #setpoints_BOOL[#tempCurrentPopup];
	    END_IF;
	    
	    //set previous values for next scan
	    #statPrevPopupIn_BOOL := #recipePopup_BOOL.IN;
	    #statPrevSetpointIn_BOOL := #setpoints_BOOL[#tempCurrentPopup].IN;
	    #statPrevPopupsSave[#INDEX_BOOL] := #recipePopup_BOOL.SaveSetpoint;
	    #statPrevPopupsRevert[#INDEX_BOOL] := #recipePopup_BOOL.RevertSetpoint;
	    
	    
	    //update main setpoint display with setpoint data
	    FOR #tempLoop := 0 TO #SETPOINTS_PERPAGE-1 DO
	        IF #tempLoop + #SETPOINTS_PERPAGE * (#recipeCurrentPages[#INDEX_BOOL] - 1) + #tempSetptsLower[#INDEX_BOOL] <= #tempSetptsUpper[#INDEX_BOOL] THEN
	            #setpointsArray_BOOL[#tempLoop] := #setpoints_BOOL[#tempLoop + #SETPOINTS_PERPAGE * (#recipeCurrentPages[#INDEX_BOOL] - 1) + #tempSetptsLower[#INDEX_BOOL]];
	            #"setpoint FaceplatesDisable_BOOL"[#tempLoop] := false;
	        ELSE
	            #"setpoint FaceplatesDisable_BOOL"[#tempLoop] := true;
	        END_IF;
	    END_FOR;
	END_REGION
	
	
	REGION STRING
	    //index in Setpoints_XXX of the current popup
	    #tempCurrentPopup := #recipePopupTrackers[#INDEX_STRING] + #SETPOINTS_PERPAGE * (#recipeCurrentPages[#INDEX_STRING] - 1) + #tempSetptsLower[#INDEX_STRING];
	    
	    IF #statPrevPopupTrackers[#INDEX_STRING] <> #recipePopupTrackers[#INDEX_STRING] THEN
	        //if a new popup has been loaded, load the new setpoint so they can be displayed
	        #recipePopup_STRING := #setpoints_STRING[#tempCurrentPopup];
	    ELSE
	        //if the HMI popup was updated, relay the commands back to the actual setpoint tag for processing
	        //taking care to ensure that changes to the setpoints tags made in other areas of the program do not get overwritten
	        IF (#statPrevPopupIn_STRING <> #recipePopup_STRING.IN) AND (#statPrevSetpointIn_STRING = #setpoints_STRING[#tempCurrentPopup].IN) THEN
	            #setpoints_STRING[#tempCurrentPopup].IN := #recipePopup_STRING.IN;
	        END_IF;
	        IF #statPrevPopupsSave[#INDEX_STRING] <> #recipePopup_STRING.SaveSetpoint THEN
	            #setpoints_STRING[#tempCurrentPopup].SaveSetpoint := #recipePopup_STRING.SaveSetpoint;
	        END_IF;
	        IF #statPrevPopupsRevert[#INDEX_STRING] <> #recipePopup_STRING.RevertSetpoint THEN
	            #setpoints_STRING[#tempCurrentPopup].RevertSetpoint := #recipePopup_STRING.RevertSetpoint;
	        END_IF;
	        
	        //then update the popup with the latest setpoint information
	        #recipePopup_STRING := #setpoints_STRING[#tempCurrentPopup];
	    END_IF;
	    
	    //set previous values for next scan
	    #statPrevPopupIn_STRING := #recipePopup_STRING.IN;
	    #statPrevSetpointIn_STRING := #setpoints_STRING[#tempCurrentPopup].IN;
	    #statPrevPopupsSave[#INDEX_STRING] := #recipePopup_STRING.SaveSetpoint;
	    #statPrevPopupsRevert[#INDEX_STRING] := #recipePopup_STRING.RevertSetpoint;
	    
	    
	    //update main setpoint display with setpoint data
	    FOR #tempLoop := 0 TO #SETPOINTS_PERPAGE - 1 DO
	        IF #tempLoop + #SETPOINTS_PERPAGE * (#recipeCurrentPages[#INDEX_STRING] - 1) + #tempSetptsLower[#INDEX_STRING] <= #tempSetptsUpper[#INDEX_STRING] THEN
	            #setpointsArray_STRING[#tempLoop] := #setpoints_STRING[#tempLoop + #SETPOINTS_PERPAGE * (#recipeCurrentPages[#INDEX_STRING] - 1) + #tempSetptsLower[#INDEX_STRING]];
	            #"setpoint FaceplatesDisable_STRING"[#tempLoop] := false;
	        ELSE
	            #"setpoint FaceplatesDisable_STRING"[#tempLoop] := true;
	        END_IF;
	    END_FOR;
	END_REGION
	
	
	REGION RECIPE NAMES AND TIMES
	    //update the recipe arrays, save times, cum times, and numbers with their current values
	    //these values are read only so no need to update the "Recipe Names Array" like we did with the popups
	    FOR #tempLoop := 0 TO #RECIPES_PERPAGE - 1 DO
	        IF #tempLoop + #RECIPES_PERPAGE * (#recipeCurrentPages[4] - 1) + #tempNumRecipesLower <= #tempNumRecipesUpper THEN
	            #recipeArrayNames[#tempLoop] := #recipeNamesArray[#tempLoop + #RECIPES_PERPAGE * (#recipeCurrentPages[4] - 1) + #tempNumRecipesLower];
	            #recipeArraySaves[#tempLoop] := #recipeSavesArray[#tempLoop + #RECIPES_PERPAGE * (#recipeCurrentPages[4] - 1) + #tempNumRecipesLower];
	            #recipeArrayTimes[#tempLoop] := #recipeTimesArray[#tempLoop + #RECIPES_PERPAGE * (#recipeCurrentPages[4] - 1) + #tempNumRecipesLower];
	            #recipeArrayNums[#tempLoop] := #tempLoop + #RECIPES_PERPAGE * (#recipeCurrentPages[4] - 1) + #tempNumRecipesLower;
	            #recipeArrayDisables[#tempLoop] := false;
	        ELSE
	            #recipeArrayDisables[#tempLoop] := true;
	        END_IF;
	    END_FOR;
	END_REGION
	
	
	
	
	
	//update previous values
	#statPrevCurrentPages := #recipeCurrentPages;
	#statPrevPopupTrackers := #recipePopupTrackers;
	
	//  -------------- END OF LOGIC -------------------------
	ENO := TRUE;   // Set the ENO output
END_FUNCTION_BLOCK

FUNCTION "LPMLV30_ConfigureDisabledUnitModes" : Void
TITLE = LPMLV30_ConfigureDisabledUnitModes
{ S7_Optimized_Access := 'TRUE' }
AUTHOR : APC_ERLF
FAMILY : OMAC
//Support: tech.team.motioncontrol@siemens.com 
//Fax: +49 (0) 9131/98-1297
   VAR_INPUT 
      ProductionModeDisable : Bool;   // TRUE: Disable unit mode Production
      MaintenanceModeDisable : Bool;   // TRUE: Disable unit mode Maintenance
      UserMode01Disable : Bool;   // TRUE: Disable user-defined unit mode 01
      UserMode02Disable : Bool;   // TRUE: Disable user-defined unit mode 02
      UserMode03Disable : Bool;   // TRUE: Disable user-defined unit mode 03
      UserMode04Disable : Bool;   // TRUE: Disable user-defined unit mode 04
      UserMode05Disable : Bool;   // TRUE: Disable user-defined unit mode 05
      UserMode06Disable : Bool;   // TRUE: Disable user-defined unit mode 06
      UserMode07Disable : Bool;   // TRUE: Disable user-defined unit mode 07
      UserMode08Disable : Bool;   // TRUE: Disable user-defined unit mode 08
   END_VAR

   VAR_OUTPUT 
      disabledUnitModes : Array[0.."LPMLV30_MAX_MODES_UPPER_LIM"] of Bool;   // Disabled unit modes configuration
   END_VAR

   VAR_TEMP 
      tempI : Int;   // Temporary Index
   END_VAR


BEGIN
	//============================================================================================================
	// SIEMENS AG
	// (c)Copyright 2015 All Rights Reserved
	//------------------------------------------------------------------------------------------------------------
	// Library: LPMLV30
	// Tested with: S7-1200 with FW version V4.1, S7-1500 with FW version V1.7
	// Engineering: TIA Portal V13 SP1
	// Restrictions: ---
	// Requirements: S7-1200 / S7-1500
	// Functionality: The function generates the unit mode configuration as Array[] of Bool.
	//------------------------------------------------------------------------------------------------------------
	// Change log table:
	// Version  Date        Expert in charge    Changes applied
	// 03.00.01 29.05.2015  RK                  First released version 
	//============================================================================================================
	// Function: LPMLV30_ConfigureDisabledUnitModes
	//============================================================================================================
	
	// Initialize unitMode configuration
	FOR #tempI := 0 TO "LPMLV30_MAX_MODES_UPPER_LIM" DO
	  #disabledUnitModes[#tempI] := TRUE;
	END_FOR;
	
	// Set unitMode configuration
	#disabledUnitModes["LPMLV30_MODE_INVALID"]     := FALSE;
	#disabledUnitModes["LPMLV30_MODE_PRODUCTION"]  := #ProductionModeDisable;
	#disabledUnitModes["LPMLV30_MODE_MAINTENANCE"] := #MaintenanceModeDisable;
	#disabledUnitModes["LPMLV30_MODE_MANUAL"]      := FALSE;
	#disabledUnitModes["LPMLV30_MODE_USER_01"]     := #UserMode01Disable;
	#disabledUnitModes["LPMLV30_MODE_USER_02"]     := #UserMode02Disable;
	#disabledUnitModes["LPMLV30_MODE_USER_03"]     := #UserMode03Disable;
	#disabledUnitModes["LPMLV30_MODE_USER_04"]     := #UserMode04Disable;
	#disabledUnitModes["LPMLV30_MODE_USER_05"]     := #UserMode05Disable;
	#disabledUnitModes["LPMLV30_MODE_USER_06"]     := #UserMode06Disable;
	#disabledUnitModes["LPMLV30_MODE_USER_07"]     := #UserMode07Disable;
	#disabledUnitModes["LPMLV30_MODE_USER_08"]     := #UserMode08Disable;
	
	//============================================================================================================
	// End of function: LPMLV30_ConfigureDisabledUnitModes
	//============================================================================================================
END_FUNCTION

FUNCTION "LPMLV30_ConfigureDisabledStates" : Void
TITLE = LPMLV30_ConfigureDisabledStates
{ S7_Optimized_Access := 'TRUE' }
AUTHOR : APC_ERLF
FAMILY : OMAC
//Support: tech.team.motioncontrol@siemens.com 
//Fax: +49 (0) 9131/98-1297
   VAR_INPUT 
      HoldingDisable : Bool;   // TRUE: Disable state Holding
      HeldDisable : Bool;   // TRUE: Disable state Held
      UnholdingDisable : Bool;   // TRUE: Disable state Unholding
      SuspendingDisable : Bool;   // TRUE: Disable state Suspending
      SuspendedDisable : Bool;   // TRUE: Disable state Suspended
      UnsuspendingDisable : Bool;   // TRUE: Disable state Unsuspending
      CompletingDisable : Bool;   // TRUE: Disable state Completing
      CompleteDisable : Bool;   // TRUE: Disable state Complete
   END_VAR

   VAR_OUTPUT 
      disabledStates : DInt;   // Disabled states configuration for one unit mode
   END_VAR

   VAR CONSTANT 
      DISABLE_ALL_STATES : DWord := 16#FFFF_FFFF;   // Disable all states
   END_VAR


BEGIN
	//============================================================================================================
	// SIEMENS AG
	// (c)Copyright 2015 All Rights Reserved
	//------------------------------------------------------------------------------------------------------------
	// Library: LPMLV30
	// Tested with: S7-1200 with FW version V4.1, S7-1500 with FW version V1.7
	// Engineering: TIA Portal V13 SP1
	// Restrictions: ---
	// Requirements: S7-1200 / S7-1500
	// Functionality: The function generates a double integer value which represents the state configuration
	//                for one unit mode.
	//------------------------------------------------------------------------------------------------------------
	// Change log table:
	// Version  Date        Expert in charge    Changes applied
	// 03.00.01 29.05.2015  RK                  First released version 
	//============================================================================================================
	// Function: LPMLV30_ConfigureDisabledStates
	//============================================================================================================
	
	#disabledStates := DWORD_TO_DINT(#DISABLE_ALL_STATES);
	
	#disabledStates.%X0  := FALSE; // Undefined state is mandatory
	#disabledStates.%X1  := FALSE; // Clearing state is mandatory
	#disabledStates.%X2  := FALSE; // Stopped state is mandatory
	#disabledStates.%X3  := FALSE; // Starting state is mandatory
	#disabledStates.%X4  := FALSE; // Idle state is mandatory
	#disabledStates.%X5  := #SuspendedDisable;
	#disabledStates.%X6  := FALSE; // Execute state is mandatory
	#disabledStates.%X7  := FALSE; // Stopping state is mandatory
	#disabledStates.%X8  := FALSE; // Aborting state is mandatory
	#disabledStates.%X9  := FALSE; // Aborted state is mandatory
	#disabledStates.%X10 := #HoldingDisable;
	#disabledStates.%X11 := #HeldDisable;
	#disabledStates.%X12 := #UnholdingDisable;
	#disabledStates.%X13 := #SuspendingDisable;
	#disabledStates.%X14 := #UnsuspendingDisable;
	#disabledStates.%X15 := FALSE; // Resetting state is mandatory
	#disabledStates.%X16 := #CompletingDisable;
	#disabledStates.%X17 := #CompleteDisable;
	
	//============================================================================================================
	// End of function: LPMLV30_ConfigureDisabledStates
	//============================================================================================================
END_FUNCTION

FUNCTION_BLOCK "EM00_00_Main"   // FB31640, LAD
TITLE = EM00_00_Main
{ S7_Optimized_Access := 'TRUE' }
AUTHOR : tech.team.motioncontrol@siemens.com
FAMILY : CPG
VERSION : 1.1
// Support: tech.team.motioncontrol@siemens.com
// stored: AutoNumber true, IsIECCheckEnabled false, IsRetainMemResEnabled false, MemoryReserve 100, SetENOAutomatically false, UDAEnableTagReadback false
   VAR
      instEventControl { ExternalAccessible := 'False'; ExternalVisible := 'False'; ExternalWritable := 'False'; S7_SetPoint := 'True'} : "EM00_01_EventControl";   // Instance DB - EM's Event Control Logic
      instPackML_ModuleSum { ExternalAccessible := 'False'; ExternalVisible := 'False'; ExternalWritable := 'False'; S7_SetPoint := 'True'} : "EM00_02_PackML_ModuleSum";   // Instance DB - EM's PackML Module Summation Logic
      instCM01 { ExternalAccessible := 'False'; ExternalVisible := 'False'; ExternalWritable := 'False'; S7_SetPoint := 'True'} : "EM00_CM01_MainOpStation";   // Instance DB - CM01
      instCM02 { ExternalAccessible := 'False'; ExternalVisible := 'False'; ExternalWritable := 'False'; S7_SetPoint := 'True'} : "EM00_CM02_Conveyor";   // Instance DB - CM02
      instCM03 { ExternalAccessible := 'False'; ExternalVisible := 'False'; ExternalWritable := 'False'; S7_SetPoint := 'True'} : "EM00_CM03_ConveyorCrossing";   // Instance DB - CM03
      instCM04 { ExternalAccessible := 'False'; ExternalVisible := 'False'; ExternalWritable := 'False'; S7_SetPoint := 'True'} : "EM00_CM04_Conveyor";   // Instance DB - CM04
      instCM05 { ExternalAccessible := 'False'; ExternalVisible := 'False'; ExternalWritable := 'False'; S7_SetPoint := 'True'} : "EM00_CM05_ConveyorCrossing";   // Instance DB - CM05
   END_VAR
   VAR_TEMP   // added for the SCL form of the ladder/FBD networks
      _w1 : Bool;
   END_VAR
BEGIN

REGION Network 1: *** BEGIN MAIN LOGIC SECTION ***
END_REGION

REGION Network 2: Call the Control Module Logic - Main Oper. Station
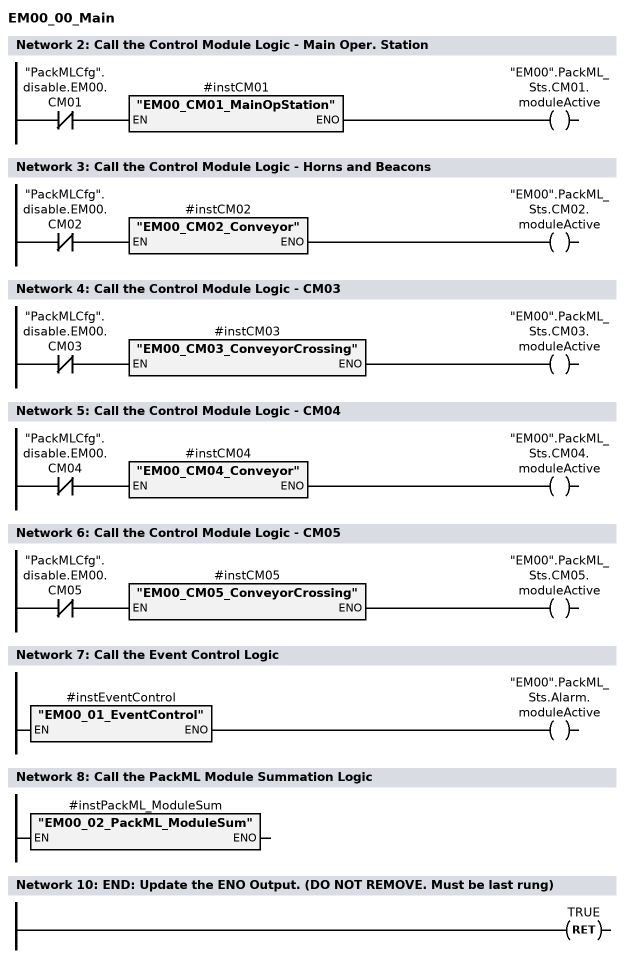
   RUNG wire#powerrail
      I_Contact( "PackMLCfg".disable.EM00.CM01 )
      #instCM01()
      Coil( "EM00".PackML_Sts.CM01.moduleActive )
   END_RUNG
   // the same network as SCL:
   #instCM01(EN := NOT "PackMLCfg".disable.EM00.CM01, ENO => #_w1);   // "EM00_CM01_MainOpStation"
   "EM00".PackML_Sts.CM01.moduleActive := #_w1;
END_REGION

REGION Network 3: Call the Control Module Logic - Horns and Beacons
   RUNG wire#powerrail
      I_Contact( "PackMLCfg".disable.EM00.CM02 )
      #instCM02()
      Coil( "EM00".PackML_Sts.CM02.moduleActive )
   END_RUNG
   // the same network as SCL:
   #instCM02(EN := NOT "PackMLCfg".disable.EM00.CM02, ENO => #_w1);   // "EM00_CM02_Conveyor"
   "EM00".PackML_Sts.CM02.moduleActive := #_w1;
END_REGION

REGION Network 4: Call the Control Module Logic - CM03
   RUNG wire#powerrail
      I_Contact( "PackMLCfg".disable.EM00.CM03 )
      #instCM03()
      Coil( "EM00".PackML_Sts.CM03.moduleActive )
   END_RUNG
   // the same network as SCL:
   #instCM03(EN := NOT "PackMLCfg".disable.EM00.CM03, ENO => #_w1);   // "EM00_CM03_ConveyorCrossing"
   "EM00".PackML_Sts.CM03.moduleActive := #_w1;
END_REGION

REGION Network 5: Call the Control Module Logic - CM04
   RUNG wire#powerrail
      I_Contact( "PackMLCfg".disable.EM00.CM04 )
      #instCM04()
      Coil( "EM00".PackML_Sts.CM04.moduleActive )
   END_RUNG
   // the same network as SCL:
   #instCM04(EN := NOT "PackMLCfg".disable.EM00.CM04, ENO => #_w1);   // "EM00_CM04_Conveyor"
   "EM00".PackML_Sts.CM04.moduleActive := #_w1;
END_REGION

REGION Network 6: Call the Control Module Logic - CM05
   RUNG wire#powerrail
      I_Contact( "PackMLCfg".disable.EM00.CM05 )
      #instCM05()
      Coil( "EM00".PackML_Sts.CM05.moduleActive )
   END_RUNG
   // the same network as SCL:
   #instCM05(EN := NOT "PackMLCfg".disable.EM00.CM05, ENO => #_w1);   // "EM00_CM05_ConveyorCrossing"
   "EM00".PackML_Sts.CM05.moduleActive := #_w1;
END_REGION

REGION Network 7: Call the Event Control Logic
   RUNG wire#powerrail
      #instEventControl()
      Coil( "EM00".PackML_Sts.Alarm.moduleActive )
   END_RUNG
   // the same network as SCL:
   #instEventControl(ENO => #_w1);   // "EM00_01_EventControl"
   "EM00".PackML_Sts.Alarm.moduleActive := #_w1;
END_REGION

REGION Network 8: Call the PackML Module Summation Logic
   RUNG wire#powerrail
      #instPackML_ModuleSum()
   END_RUNG
   // the same network as SCL:
   #instPackML_ModuleSum();   // "EM00_02_PackML_ModuleSum"
END_REGION

REGION Network 10: END: Update the ENO Output. (DO NOT REMOVE. Must be last rung)
   RUNG wire#powerrail
      ReturnCoil( TRUE )
   END_RUNG
   // the same network as SCL:
   ENO := TRUE;
   RETURN;
END_REGION
END_FUNCTION_BLOCK

FUNCTION_BLOCK "EM00_CM01_MainOpStation"   // FB31651, LAD
TITLE = EM00_CM01_MainOpStation
{ S7_Optimized_Access := 'TRUE' }
AUTHOR : tech.team.motioncontrol@siemens.com
FAMILY : CPG
VERSION : 1.1
// Support: tech.team.motioncontrol@siemens.com
// stored: AutoNumber true, IsIECCheckEnabled false, IsRetainMemResEnabled false, MemoryReserve 100, SetENOAutomatically false, UDAEnableTagReadback false
   VAR
      instAlarm_EStop { ExternalAccessible := 'False'; ExternalVisible := 'False'; ExternalWritable := 'False'; S7_SetPoint := 'True'} : "CPG_Event";   // Alarm Event - EStop pressed (Event instance)
      instAlarm_HMI_StopPB { ExternalAccessible := 'False'; ExternalVisible := 'False'; ExternalWritable := 'False'; S7_SetPoint := 'True'} : "CPG_Event";   // Alarm Event - HMI Stop PB pressed (Event instance)
      instStatus_WaitingForStartCmd { ExternalAccessible := 'False'; ExternalVisible := 'False'; ExternalWritable := 'False'; S7_SetPoint := 'True'} : "CPG_Event";   // Status Event - waiting for start command (Event instance)
      instStatus_WaitingForResetCmd { ExternalAccessible := 'False'; ExternalVisible := 'False'; ExternalWritable := 'False'; S7_SetPoint := 'True'} : "CPG_Event";   // Status Event - waiting for reset command (Event instance)
      instAlarm_Hold_PB { ExternalAccessible := 'False'; ExternalVisible := 'False'; ExternalWritable := 'False'; S7_SetPoint := 'True'} : "CPG_Event";   // Alarm Event - HMI Held PB pressed (Event instance)
      instStatus_WaitingForUnHoldCmd { ExternalAccessible := 'False'; ExternalVisible := 'False'; ExternalWritable := 'False'; S7_SetPoint := 'True'} : "CPG_Event";   // Status Event - waiting for unhold command (Event instance)
      instTimer_StartingDelay_SC { ExternalAccessible := 'False'; ExternalVisible := 'False'; ExternalWritable := 'False'; S7_SetPoint := 'True'} : IEC_TIMER;   // IEC Timer - starting delay (demo only - used to slow state model transition)
      instTimer_CompletingDelay_SC { ExternalAccessible := 'False'; ExternalVisible := 'False'; ExternalWritable := 'False'; S7_SetPoint := 'True'} : IEC_TIMER;   // IEC Timer - completing delay (demo only - used to slow state model transition)
      instTimer_AbortingDelay_SC { ExternalAccessible := 'False'; ExternalVisible := 'False'; ExternalWritable := 'False'; S7_SetPoint := 'True'} : IEC_TIMER;   // IEC Timer - aborting delay (demo only - used to slow state model transition)
      instTimer_StoppingDelay_SC { ExternalAccessible := 'False'; ExternalVisible := 'False'; ExternalWritable := 'False'; S7_SetPoint := 'True'} : IEC_TIMER;   // IEC Timer - stopping delay (demo only - used to slow state model transition)
      instTimer_ResettingDelay_SC { ExternalAccessible := 'False'; ExternalVisible := 'False'; ExternalWritable := 'False'; S7_SetPoint := 'True'} : IEC_TIMER;   // IEC Timer - resetting delay (demo only - used to slow state model transition)
      instTimer_HoldingDelay_SC { ExternalAccessible := 'False'; ExternalVisible := 'False'; ExternalWritable := 'False'; S7_SetPoint := 'True'} : IEC_TIMER;   // IEC Timer - holding delay (demo only - used to slow state model transition)
      instTimer_UnHoldingDelay_SC { ExternalAccessible := 'False'; ExternalVisible := 'False'; ExternalWritable := 'False'; S7_SetPoint := 'True'} : IEC_TIMER;   // IEC Timer - un-holding delay (demo only - used to slow state model transition)
      instTimer_SuspendingDelay_SC { ExternalAccessible := 'False'; ExternalVisible := 'False'; ExternalWritable := 'False'; S7_SetPoint := 'True'} : IEC_TIMER;   // IEC Timer - suspending delay (demo only - used to slow state model transition)
      instTimer_UnSuspendingDelay_SC { ExternalAccessible := 'False'; ExternalVisible := 'False'; ExternalWritable := 'False'; S7_SetPoint := 'True'} : IEC_TIMER;   // IEC Timer - un-suspending delay (demo only - used to slow state model transition)
      instTimer_ClearingDelay_SC { ExternalAccessible := 'False'; ExternalVisible := 'False'; ExternalWritable := 'False'; S7_SetPoint := 'True'} : IEC_TIMER;   // IEC Timer - clearing delay (demo only - used to slow state model transition)
   END_VAR
BEGIN

REGION Network 1: *** Begin the Setpoint Management Information Section ***
END_REGION

REGION Network 2: *** Begin the Logic Section ***
END_REGION

REGION Network 3: *** Begin the Event Information Section ***
END_REGION

REGION Network 4: Alarm Event - EStop
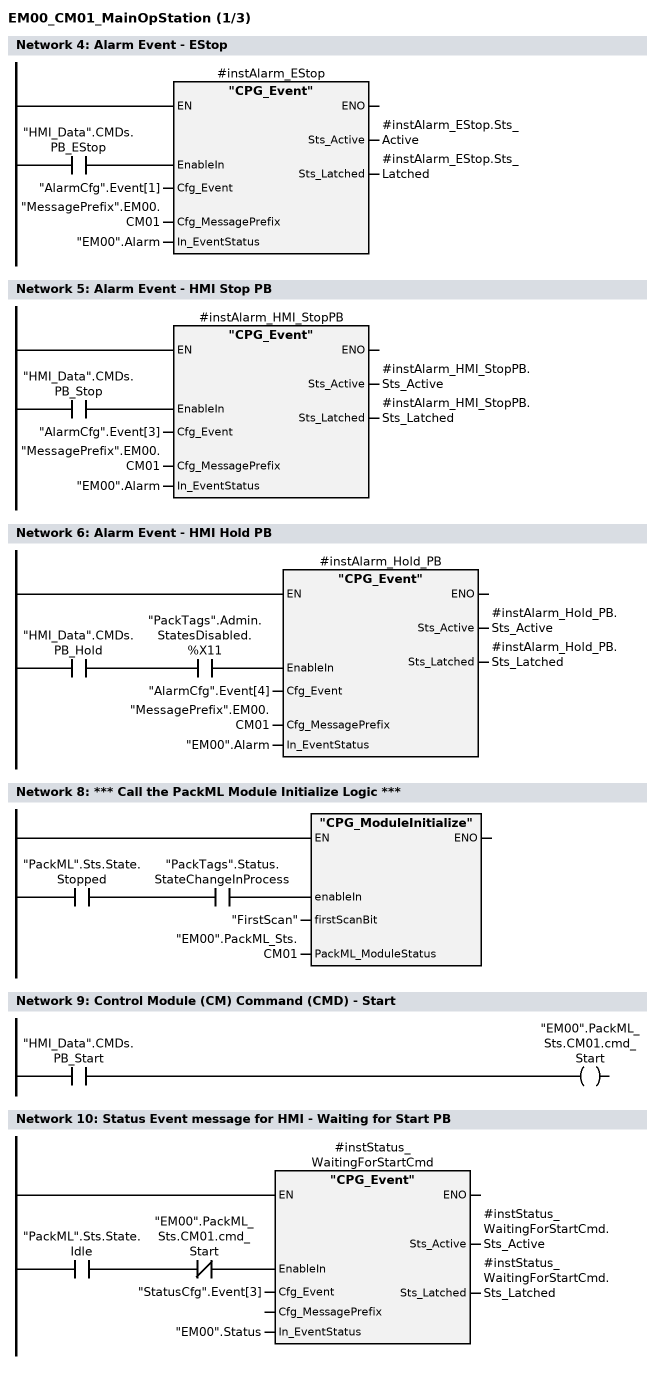
   RUNG wire#powerrail
      #instAlarm_EStop(EnableIn := wire#w1, Cfg_Event := "AlarmCfg".Event[1], Cfg_MessagePrefix := "MessagePrefix".EM00.CM01, In_EventStatus := "EM00".Alarm, Sts_Active => #instAlarm_EStop.Sts_Active, Sts_Latched => #instAlarm_EStop.Sts_Latched)
   END_RUNG
   RUNG wire#powerrail
      Contact( "HMI_Data".CMDs.PB_EStop )
   END_RUNG wire#w1
   // the same network as SCL:
   #instAlarm_EStop(EnableIn := "HMI_Data".CMDs.PB_EStop,   // "CPG_Event"
                    Cfg_Event := "AlarmCfg".Event[1],
                    Cfg_MessagePrefix := "MessagePrefix".EM00.CM01,
                    In_EventStatus := "EM00".Alarm,
                    Sts_Active => #instAlarm_EStop.Sts_Active,
                    Sts_Latched => #instAlarm_EStop.Sts_Latched);
END_REGION

REGION Network 5: Alarm Event - HMI Stop PB
   RUNG wire#powerrail
      #instAlarm_HMI_StopPB(EnableIn := wire#w1, Cfg_Event := "AlarmCfg".Event[3], Cfg_MessagePrefix := "MessagePrefix".EM00.CM01, In_EventStatus := "EM00".Alarm, Sts_Active => #instAlarm_HMI_StopPB.Sts_Active, Sts_Latched => #instAlarm_HMI_StopPB.Sts_Latched)
   END_RUNG
   RUNG wire#powerrail
      Contact( "HMI_Data".CMDs.PB_Stop )
   END_RUNG wire#w1
   // the same network as SCL:
   #instAlarm_HMI_StopPB(EnableIn := "HMI_Data".CMDs.PB_Stop,   // "CPG_Event"
                         Cfg_Event := "AlarmCfg".Event[3],
                         Cfg_MessagePrefix := "MessagePrefix".EM00.CM01,
                         In_EventStatus := "EM00".Alarm,
                         Sts_Active => #instAlarm_HMI_StopPB.Sts_Active,
                         Sts_Latched => #instAlarm_HMI_StopPB.Sts_Latched);
END_REGION

REGION Network 6: Alarm Event - HMI Hold PB
   RUNG wire#powerrail
      #instAlarm_Hold_PB(EnableIn := wire#w1, Cfg_Event := "AlarmCfg".Event[4], Cfg_MessagePrefix := "MessagePrefix".EM00.CM01, In_EventStatus := "EM00".Alarm, Sts_Active => #instAlarm_Hold_PB.Sts_Active, Sts_Latched => #instAlarm_Hold_PB.Sts_Latched)
   END_RUNG
   RUNG wire#powerrail
      Contact( "HMI_Data".CMDs.PB_Hold )
      Contact( "PackTags".Admin.StatesDisabled.%X11 )
   END_RUNG wire#w1
   // the same network as SCL:
   #instAlarm_Hold_PB(EnableIn := "HMI_Data".CMDs.PB_Hold AND "PackTags".Admin.StatesDisabled.%X11,   // "CPG_Event"
                      Cfg_Event := "AlarmCfg".Event[4],
                      Cfg_MessagePrefix := "MessagePrefix".EM00.CM01,
                      In_EventStatus := "EM00".Alarm,
                      Sts_Active => #instAlarm_Hold_PB.Sts_Active,
                      Sts_Latched => #instAlarm_Hold_PB.Sts_Latched);
END_REGION

REGION Network 7: *** Begin the State Model Status Feedback Section ***
END_REGION

REGION Network 8: *** Call the PackML Module Initialize Logic ***
   RUNG wire#powerrail
      "CPG_ModuleInitialize"(enableIn := wire#w1, firstScanBit := "FirstScan", PackML_ModuleStatus := "EM00".PackML_Sts.CM01)
   END_RUNG
   RUNG wire#powerrail
      Contact( "PackML".Sts.State.Stopped )
      Contact( "PackTags".Status.StateChangeInProcess )
   END_RUNG wire#w1
   // the same network as SCL:
   "CPG_ModuleInitialize"(enableIn := "PackML".Sts.State.Stopped AND "PackTags".Status.StateChangeInProcess,
                          firstScanBit := "FirstScan",
                          PackML_ModuleStatus := "EM00".PackML_Sts.CM01);
END_REGION

REGION Network 9: Control Module (CM) Command (CMD) - Start
   RUNG wire#powerrail
      Contact( "HMI_Data".CMDs.PB_Start )
      Coil( "EM00".PackML_Sts.CM01.cmd_Start )
   END_RUNG
   // the same network as SCL:
   "EM00".PackML_Sts.CM01.cmd_Start := "HMI_Data".CMDs.PB_Start;
END_REGION

REGION Network 10: Status Event message for HMI - Waiting for Start PB
   RUNG wire#powerrail
      #instStatus_WaitingForStartCmd(EnableIn := wire#w1, Cfg_Event := "StatusCfg".Event[3], Cfg_MessagePrefix :=, In_EventStatus := "EM00".Status, Sts_Active => #instStatus_WaitingForStartCmd.Sts_Active, Sts_Latched => #instStatus_WaitingForStartCmd.Sts_Latched)
   END_RUNG
   RUNG wire#powerrail
      Contact( "PackML".Sts.State.Idle )
      I_Contact( "EM00".PackML_Sts.CM01.cmd_Start )
   END_RUNG wire#w1
   // the same network as SCL:
   #instStatus_WaitingForStartCmd(EnableIn := "PackML".Sts.State.Idle AND NOT "EM00".PackML_Sts.CM01.cmd_Start,   // "CPG_Event"
                           Cfg_Event := "StatusCfg".Event[3],
                           In_EventStatus := "EM00".Status,
                           Sts_Active => #instStatus_WaitingForStartCmd.Sts_Active,
                           Sts_Latched => #instStatus_WaitingForStartCmd.Sts_Latched);
END_REGION

REGION Network 11: Control Module (CM) Command (CMD) - reset and clear commands
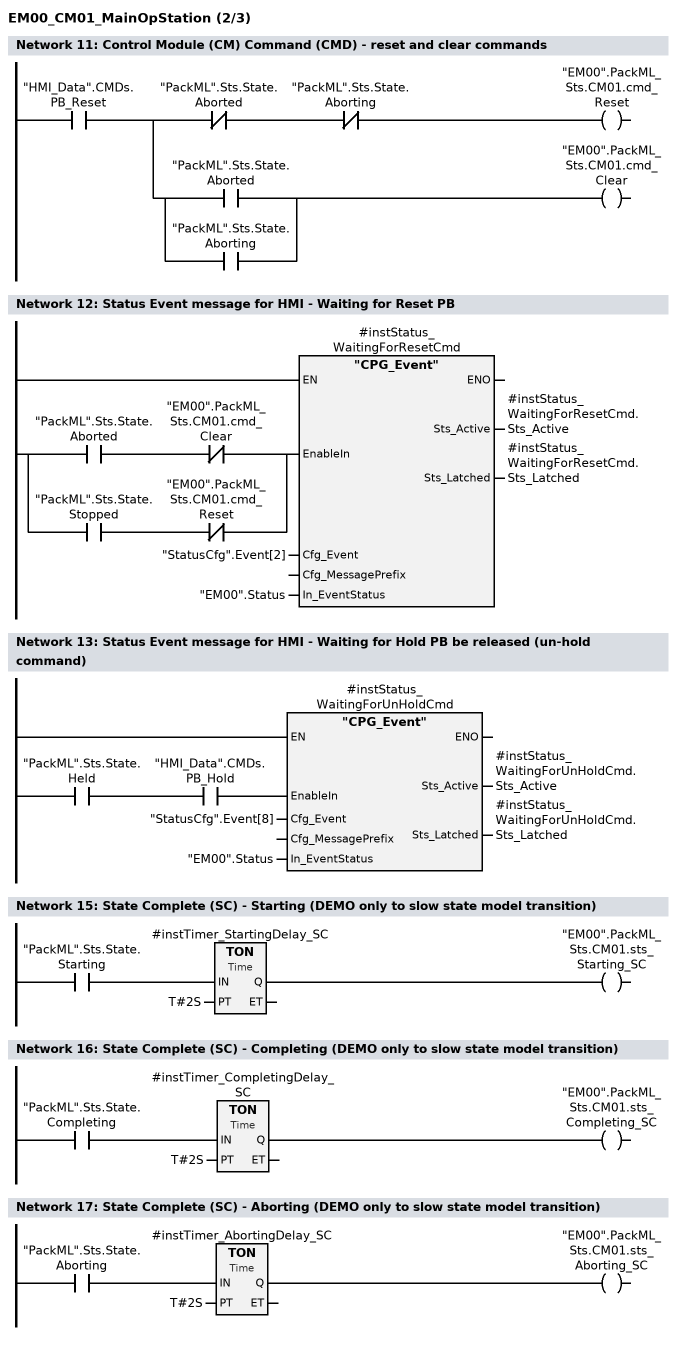
   RUNG wire#powerrail
      Contact( "HMI_Data".CMDs.PB_Reset )
      wire#w1
      I_Contact( "PackML".Sts.State.Aborted )
      I_Contact( "PackML".Sts.State.Aborting )
      Coil( "EM00".PackML_Sts.CM01.cmd_Reset )
   END_RUNG
   RUNG wire#w1
      Contact( "PackML".Sts.State.Aborted )
      wire#w2
      Coil( "EM00".PackML_Sts.CM01.cmd_Clear )
   END_RUNG
   RUNG wire#w1
      Contact( "PackML".Sts.State.Aborting )
   END_RUNG wire#w2
   // the same network as SCL:
   "EM00".PackML_Sts.CM01.cmd_Reset := "HMI_Data".CMDs.PB_Reset AND NOT "PackML".Sts.State.Aborted AND NOT "PackML".Sts.State.Aborting;
   "EM00".PackML_Sts.CM01.cmd_Clear := "HMI_Data".CMDs.PB_Reset AND ("PackML".Sts.State.Aborted OR "PackML".Sts.State.Aborting);
END_REGION

REGION Network 12: Status Event message for HMI - Waiting for Reset PB
   RUNG wire#powerrail
      #instStatus_WaitingForResetCmd(EnableIn := wire#w1, Cfg_Event := "StatusCfg".Event[2], Cfg_MessagePrefix :=, In_EventStatus := "EM00".Status, Sts_Active => #instStatus_WaitingForResetCmd.Sts_Active, Sts_Latched => #instStatus_WaitingForResetCmd.Sts_Latched)
   END_RUNG
   RUNG wire#powerrail
      Contact( "PackML".Sts.State.Aborted )
      I_Contact( "EM00".PackML_Sts.CM01.cmd_Clear )
   END_RUNG wire#w1
   RUNG wire#powerrail
      Contact( "PackML".Sts.State.Stopped )
      I_Contact( "EM00".PackML_Sts.CM01.cmd_Reset )
   END_RUNG wire#w1
   // the same network as SCL:
   #instStatus_WaitingForResetCmd(EnableIn := ("PackML".Sts.State.Aborted AND NOT "EM00".PackML_Sts.CM01.cmd_Clear) OR ("PackML".Sts.State.Stopped AND NOT "EM00".PackML_Sts.CM01.cmd_Reset),   // "CPG_Event"
                           Cfg_Event := "StatusCfg".Event[2],
                           In_EventStatus := "EM00".Status,
                           Sts_Active => #instStatus_WaitingForResetCmd.Sts_Active,
                           Sts_Latched => #instStatus_WaitingForResetCmd.Sts_Latched);
END_REGION

REGION Network 13: Status Event message for HMI - Waiting for Hold PB be released (un-hold command)
   RUNG wire#powerrail
      #instStatus_WaitingForUnHoldCmd(EnableIn := wire#w1, Cfg_Event := "StatusCfg".Event[8], Cfg_MessagePrefix :=, In_EventStatus := "EM00".Status, Sts_Active => #instStatus_WaitingForUnHoldCmd.Sts_Active, Sts_Latched => #instStatus_WaitingForUnHoldCmd.Sts_Latched)
   END_RUNG
   RUNG wire#powerrail
      Contact( "PackML".Sts.State.Held )
      Contact( "HMI_Data".CMDs.PB_Hold )
   END_RUNG wire#w1
   // the same network as SCL:
   #instStatus_WaitingForUnHoldCmd(EnableIn := "PackML".Sts.State.Held AND "HMI_Data".CMDs.PB_Hold,   // "CPG_Event"
                           Cfg_Event := "StatusCfg".Event[8],
                           In_EventStatus := "EM00".Status,
                           Sts_Active => #instStatus_WaitingForUnHoldCmd.Sts_Active,
                           Sts_Latched => #instStatus_WaitingForUnHoldCmd.Sts_Latched);
END_REGION

REGION Network 14: State Model delay timers used to slow state model transition - only used for demo purposes (remove for real projects)
END_REGION

REGION Network 15: State Complete (SC) - Starting (DEMO only to slow state model transition)
   RUNG wire#powerrail
      Contact( "PackML".Sts.State.Starting )
      { S7_Templates := "time_type := Time" } #instTimer_StartingDelay_SC.TON(pt := T#2S, et =>)
      Coil( "EM00".PackML_Sts.CM01.sts_Starting_SC )
   END_RUNG
   // the same network as SCL:
   #instTimer_StartingDelay_SC.TON(IN := "PackML".Sts.State.Starting, PT := T#2S);
   "EM00".PackML_Sts.CM01.sts_Starting_SC := #instTimer_StartingDelay_SC.Q;
END_REGION

REGION Network 16: State Complete (SC) - Completing (DEMO only to slow state model transition)
   RUNG wire#powerrail
      Contact( "PackML".Sts.State.Completing )
      { S7_Templates := "time_type := Time" } #instTimer_CompletingDelay_SC.TON(pt := T#2S, et =>)
      Coil( "EM00".PackML_Sts.CM01.sts_Completing_SC )
   END_RUNG
   // the same network as SCL:
   #instTimer_CompletingDelay_SC.TON(IN := "PackML".Sts.State.Completing, PT := T#2S);
   "EM00".PackML_Sts.CM01.sts_Completing_SC := #instTimer_CompletingDelay_SC.Q;
END_REGION

REGION Network 17: State Complete (SC) - Aborting (DEMO only to slow state model transition)
   RUNG wire#powerrail
      Contact( "PackML".Sts.State.Aborting )
      { S7_Templates := "time_type := Time" } #instTimer_AbortingDelay_SC.TON(pt := T#2S, et =>)
      Coil( "EM00".PackML_Sts.CM01.sts_Aborting_SC )
   END_RUNG
   // the same network as SCL:
   #instTimer_AbortingDelay_SC.TON(IN := "PackML".Sts.State.Aborting, PT := T#2S);
   "EM00".PackML_Sts.CM01.sts_Aborting_SC := #instTimer_AbortingDelay_SC.Q;
END_REGION

REGION Network 18: State Complete (SC) - Stopping (DEMO only to slow state model transition)
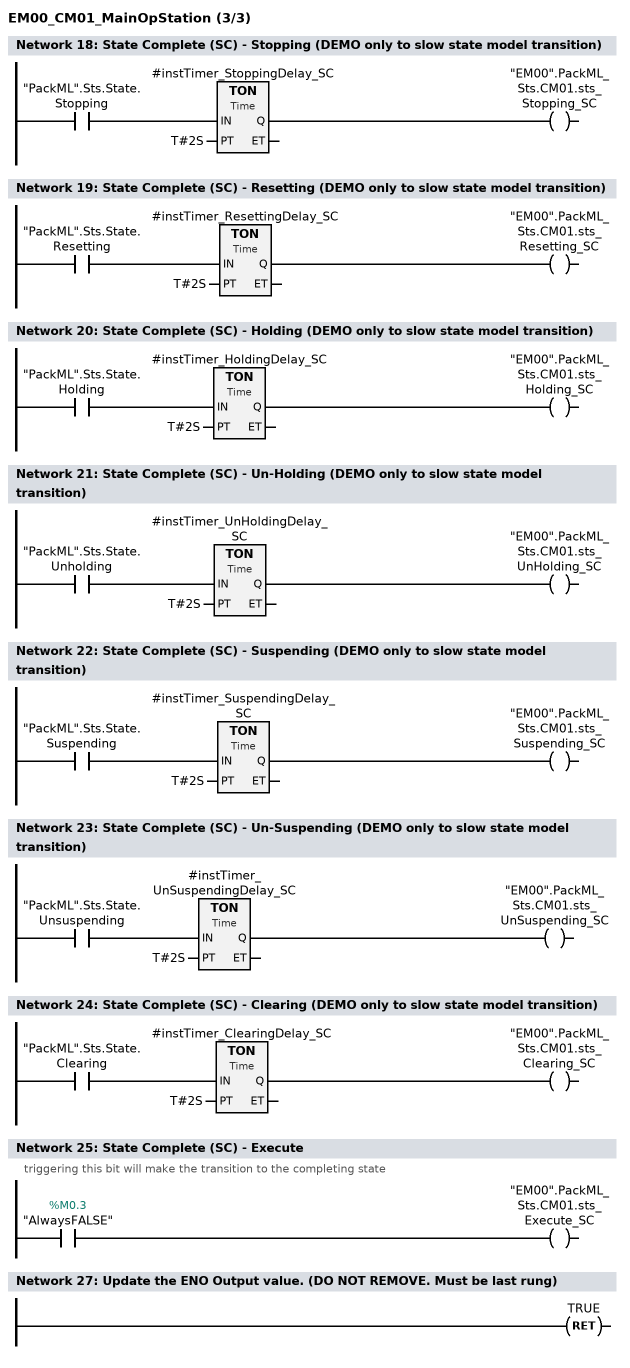
   RUNG wire#powerrail
      Contact( "PackML".Sts.State.Stopping )
      { S7_Templates := "time_type := Time" } #instTimer_StoppingDelay_SC.TON(pt := T#2S, et =>)
      Coil( "EM00".PackML_Sts.CM01.sts_Stopping_SC )
   END_RUNG
   // the same network as SCL:
   #instTimer_StoppingDelay_SC.TON(IN := "PackML".Sts.State.Stopping, PT := T#2S);
   "EM00".PackML_Sts.CM01.sts_Stopping_SC := #instTimer_StoppingDelay_SC.Q;
END_REGION

REGION Network 19: State Complete (SC) - Resetting (DEMO only to slow state model transition)
   RUNG wire#powerrail
      Contact( "PackML".Sts.State.Resetting )
      { S7_Templates := "time_type := Time" } #instTimer_ResettingDelay_SC.TON(pt := T#2S, et =>)
      Coil( "EM00".PackML_Sts.CM01.sts_Resetting_SC )
   END_RUNG
   // the same network as SCL:
   #instTimer_ResettingDelay_SC.TON(IN := "PackML".Sts.State.Resetting, PT := T#2S);
   "EM00".PackML_Sts.CM01.sts_Resetting_SC := #instTimer_ResettingDelay_SC.Q;
END_REGION

REGION Network 20: State Complete (SC) - Holding (DEMO only to slow state model transition)
   RUNG wire#powerrail
      Contact( "PackML".Sts.State.Holding )
      { S7_Templates := "time_type := Time" } #instTimer_HoldingDelay_SC.TON(pt := T#2S, et =>)
      Coil( "EM00".PackML_Sts.CM01.sts_Holding_SC )
   END_RUNG
   // the same network as SCL:
   #instTimer_HoldingDelay_SC.TON(IN := "PackML".Sts.State.Holding, PT := T#2S);
   "EM00".PackML_Sts.CM01.sts_Holding_SC := #instTimer_HoldingDelay_SC.Q;
END_REGION

REGION Network 21: State Complete (SC) - Un-Holding (DEMO only to slow state model transition)
   RUNG wire#powerrail
      Contact( "PackML".Sts.State.Unholding )
      { S7_Templates := "time_type := Time" } #instTimer_UnHoldingDelay_SC.TON(pt := T#2S, et =>)
      Coil( "EM00".PackML_Sts.CM01.sts_UnHolding_SC )
   END_RUNG
   // the same network as SCL:
   #instTimer_UnHoldingDelay_SC.TON(IN := "PackML".Sts.State.Unholding, PT := T#2S);
   "EM00".PackML_Sts.CM01.sts_UnHolding_SC := #instTimer_UnHoldingDelay_SC.Q;
END_REGION

REGION Network 22: State Complete (SC) - Suspending (DEMO only to slow state model transition)
   RUNG wire#powerrail
      Contact( "PackML".Sts.State.Suspending )
      { S7_Templates := "time_type := Time" } #instTimer_SuspendingDelay_SC.TON(pt := T#2S, et =>)
      Coil( "EM00".PackML_Sts.CM01.sts_Suspending_SC )
   END_RUNG
   // the same network as SCL:
   #instTimer_SuspendingDelay_SC.TON(IN := "PackML".Sts.State.Suspending, PT := T#2S);
   "EM00".PackML_Sts.CM01.sts_Suspending_SC := #instTimer_SuspendingDelay_SC.Q;
END_REGION

REGION Network 23: State Complete (SC) - Un-Suspending (DEMO only to slow state model transition)
   RUNG wire#powerrail
      Contact( "PackML".Sts.State.Unsuspending )
      { S7_Templates := "time_type := Time" } #instTimer_UnSuspendingDelay_SC.TON(pt := T#2S, et =>)
      Coil( "EM00".PackML_Sts.CM01.sts_UnSuspending_SC )
   END_RUNG
   // the same network as SCL:
   #instTimer_UnSuspendingDelay_SC.TON(IN := "PackML".Sts.State.Unsuspending, PT := T#2S);
   "EM00".PackML_Sts.CM01.sts_UnSuspending_SC := #instTimer_UnSuspendingDelay_SC.Q;
END_REGION

REGION Network 24: State Complete (SC) - Clearing (DEMO only to slow state model transition)
   RUNG wire#powerrail
      Contact( "PackML".Sts.State.Clearing )
      { S7_Templates := "time_type := Time" } #instTimer_ClearingDelay_SC.TON(pt := T#2S, et =>)
      Coil( "EM00".PackML_Sts.CM01.sts_Clearing_SC )
   END_RUNG
   // the same network as SCL:
   #instTimer_ClearingDelay_SC.TON(IN := "PackML".Sts.State.Clearing, PT := T#2S);
   "EM00".PackML_Sts.CM01.sts_Clearing_SC := #instTimer_ClearingDelay_SC.Q;
END_REGION

REGION Network 25: State Complete (SC) - Execute
   // triggering this bit will make the transition to the completing state
   RUNG wire#powerrail
      Contact( "AlwaysFALSE" )
      Coil( "EM00".PackML_Sts.CM01.sts_Execute_SC )
   END_RUNG
   // the same network as SCL:
   "EM00".PackML_Sts.CM01.sts_Execute_SC := "AlwaysFALSE";
END_REGION

REGION Network 27: Update the ENO Output value. (DO NOT REMOVE. Must be last rung)
   RUNG wire#powerrail
      ReturnCoil( TRUE )
   END_RUNG
   // the same network as SCL:
   ENO := TRUE;
   RETURN;
END_REGION
END_FUNCTION_BLOCK

FUNCTION_BLOCK "EM00_CM02_Conveyor"   // FB31652, LAD
TITLE = EM00_CM02_HornBeacons
{ S7_Optimized_Access := 'TRUE' }
AUTHOR : tech.team.motioncontrol@siemens.com
FAMILY : CPG
VERSION : 1.1
// Support: tech.team.motioncontrol@siemens.com
// stored: AutoNumber true, IsIECCheckEnabled false, IsRetainMemResEnabled false, MemoryReserve 100, SetENOAutomatically false, UDAEnableTagReadback false
   VAR
      statDummy { ExternalAccessible := 'False'; ExternalVisible := 'False'; ExternalWritable := 'False'} : Bool;   // Variable to control a horn
   END_VAR
BEGIN

REGION Network 1: *** Begin the Setpoint Management Information Section ***
END_REGION

REGION Network 2: *** Begin the Logic Section ***
END_REGION

REGION Network 3: Horn delay timer - startup
END_REGION

REGION Network 4: *** Begin the Event Information Section ***
END_REGION

REGION Network 5: *** Begin the State Model Status Feedback Section ***
END_REGION

REGION Network 6: *** Call the PackML Module Initialize Logic ***
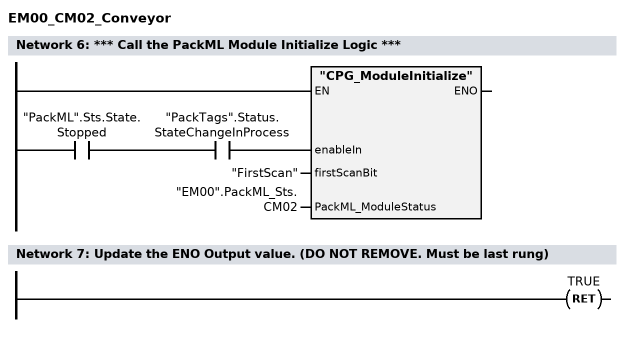
   RUNG wire#powerrail
      "CPG_ModuleInitialize"(enableIn := wire#w1, firstScanBit := "FirstScan", PackML_ModuleStatus := "EM00".PackML_Sts.CM02)
   END_RUNG
   RUNG wire#powerrail
      Contact( "PackML".Sts.State.Stopped )
      Contact( "PackTags".Status.StateChangeInProcess )
   END_RUNG wire#w1
   // the same network as SCL:
   "CPG_ModuleInitialize"(enableIn := "PackML".Sts.State.Stopped AND "PackTags".Status.StateChangeInProcess,
                          firstScanBit := "FirstScan",
                          PackML_ModuleStatus := "EM00".PackML_Sts.CM02);
END_REGION

REGION Network 7: Update the ENO Output value. (DO NOT REMOVE. Must be last rung)
   RUNG wire#powerrail
      ReturnCoil( TRUE )
   END_RUNG
   // the same network as SCL:
   ENO := TRUE;
   RETURN;
END_REGION
END_FUNCTION_BLOCK

FUNCTION_BLOCK "EM00_CM03_ConveyorCrossing"   // FB31653, LAD
TITLE = EM00_CM03
{ S7_Optimized_Access := 'TRUE' }
AUTHOR : tech.team.motioncontrol@siemens.com
FAMILY : CPG
VERSION : 1.1
// Support: tech.team.motioncontrol@siemens.com
// stored: AutoNumber true, IsIECCheckEnabled false, IsRetainMemResEnabled false, MemoryReserve 100, SetENOAutomatically false, UDAEnableTagReadback false
   VAR
      statDummyBool { ExternalAccessible := 'False'; ExternalVisible := 'False'; ExternalWritable := 'False'} : Bool;   // dummy bool - placeholder
   END_VAR
BEGIN

REGION Network 1: *** Begin the Setpoint Management Information Section ***
END_REGION

REGION Network 2: *** Begin the Logic Section ***
END_REGION

REGION Network 3: *** Begin the Event Information Section ***
END_REGION

REGION Network 4: *** Begin the State Model Status Feedback Section ***
END_REGION

REGION Network 5: *** Call the PackML Module Initialize Logic ***
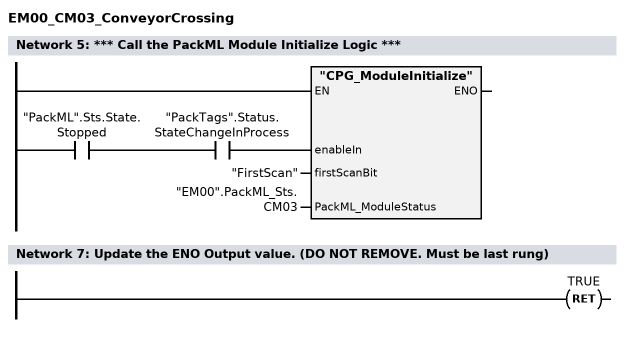
   RUNG wire#powerrail
      "CPG_ModuleInitialize"(enableIn := wire#w1, firstScanBit := "FirstScan", PackML_ModuleStatus := "EM00".PackML_Sts.CM03)
   END_RUNG
   RUNG wire#powerrail
      Contact( "PackML".Sts.State.Stopped )
      Contact( "PackTags".Status.StateChangeInProcess )
   END_RUNG wire#w1
   // the same network as SCL:
   "CPG_ModuleInitialize"(enableIn := "PackML".Sts.State.Stopped AND "PackTags".Status.StateChangeInProcess,
                          firstScanBit := "FirstScan",
                          PackML_ModuleStatus := "EM00".PackML_Sts.CM03);
END_REGION

REGION Network 7: Update the ENO Output value. (DO NOT REMOVE. Must be last rung)
   RUNG wire#powerrail
      ReturnCoil( TRUE )
   END_RUNG
   // the same network as SCL:
   ENO := TRUE;
   RETURN;
END_REGION
END_FUNCTION_BLOCK

FUNCTION_BLOCK "EM00_CM04_Conveyor"   // FB31654, LAD
TITLE = EM00_CM04
{ S7_Optimized_Access := 'TRUE' }
AUTHOR : tech.team.motioncontrol@siemens.com
FAMILY : CPG
VERSION : 1.1
// Support: tech.team.motioncontrol@siemens.com
// stored: AutoNumber true, IsIECCheckEnabled false, IsRetainMemResEnabled false, MemoryReserve 100, SetENOAutomatically false, UDAEnableTagReadback false
   VAR
      statDummyBool { ExternalAccessible := 'False'; ExternalVisible := 'False'; ExternalWritable := 'False'} : Bool;   // dummy bool - placeholder
   END_VAR
BEGIN

REGION Network 1: *** Begin the Setpoint Management Information Section ***
END_REGION

REGION Network 2: *** Begin the Logic Section ***
END_REGION

REGION Network 3: *** Begin the Event Information Section ***
END_REGION

REGION Network 4: *** Begin the State Model Status Feedback Section ***
END_REGION

REGION Network 5: *** Call the PackML Module Initialize Logic ***
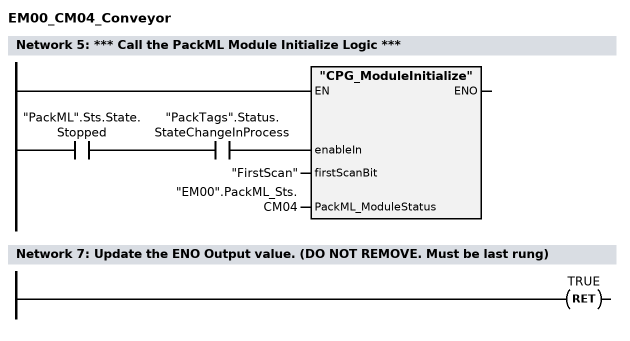
   RUNG wire#powerrail
      "CPG_ModuleInitialize"(enableIn := wire#w1, firstScanBit := "FirstScan", PackML_ModuleStatus := "EM00".PackML_Sts.CM04)
   END_RUNG
   RUNG wire#powerrail
      Contact( "PackML".Sts.State.Stopped )
      Contact( "PackTags".Status.StateChangeInProcess )
   END_RUNG wire#w1
   // the same network as SCL:
   "CPG_ModuleInitialize"(enableIn := "PackML".Sts.State.Stopped AND "PackTags".Status.StateChangeInProcess,
                          firstScanBit := "FirstScan",
                          PackML_ModuleStatus := "EM00".PackML_Sts.CM04);
END_REGION

REGION Network 7: Update the ENO Output value. (DO NOT REMOVE. Must be last rung)
   RUNG wire#powerrail
      ReturnCoil( TRUE )
   END_RUNG
   // the same network as SCL:
   ENO := TRUE;
   RETURN;
END_REGION
END_FUNCTION_BLOCK

FUNCTION_BLOCK "EM00_CM05_ConveyorCrossing"   // FB31655, LAD
TITLE = EM00_CM05
{ S7_Optimized_Access := 'TRUE' }
AUTHOR : tech.team.motioncontrol@siemens.com
FAMILY : CPG
VERSION : 1.1
// Support: tech.team.motioncontrol@siemens.com
// stored: AutoNumber true, IsIECCheckEnabled false, IsRetainMemResEnabled false, MemoryReserve 100, SetENOAutomatically false, UDAEnableTagReadback false
   VAR
      statDummyBool { ExternalAccessible := 'False'; ExternalVisible := 'False'; ExternalWritable := 'False'} : Bool;   // dummy bool - placeholder
   END_VAR
BEGIN

REGION Network 1: *** Begin the Setpoint Management Information Section ***
END_REGION

REGION Network 2: *** Begin the Logic Section ***
END_REGION

REGION Network 3: *** Begin the Event Information Section ***
END_REGION

REGION Network 4: *** Begin the State Model Status Feedback Section ***
END_REGION

REGION Network 5: *** Call the PackML Module Initialize Logic ***
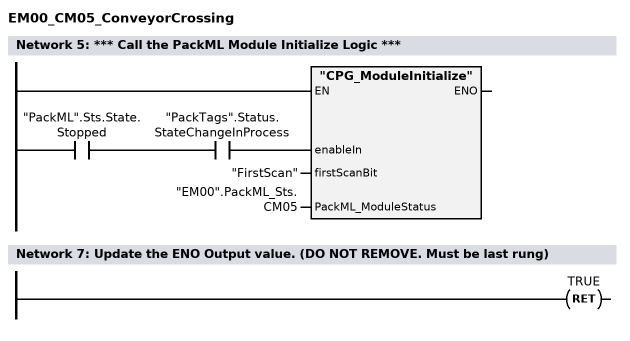
   RUNG wire#powerrail
      "CPG_ModuleInitialize"(enableIn := wire#w1, firstScanBit := "FirstScan", PackML_ModuleStatus := "EM00".PackML_Sts.CM05)
   END_RUNG
   RUNG wire#powerrail
      Contact( "PackML".Sts.State.Stopped )
      Contact( "PackTags".Status.StateChangeInProcess )
   END_RUNG wire#w1
   // the same network as SCL:
   "CPG_ModuleInitialize"(enableIn := "PackML".Sts.State.Stopped AND "PackTags".Status.StateChangeInProcess,
                          firstScanBit := "FirstScan",
                          PackML_ModuleStatus := "EM00".PackML_Sts.CM05);
END_REGION

REGION Network 7: Update the ENO Output value. (DO NOT REMOVE. Must be last rung)
   RUNG wire#powerrail
      ReturnCoil( TRUE )
   END_RUNG
   // the same network as SCL:
   ENO := TRUE;
   RETURN;
END_REGION
END_FUNCTION_BLOCK

FUNCTION_BLOCK "EM00_01_EventControl"   // FB31641, LAD
TITLE = EM00_01_EventControl
{ S7_Optimized_Access := 'TRUE' }
AUTHOR : tech.team.motioncontrol@siemens.com
FAMILY : CPG
VERSION : 1.1
// Support: tech.team.motioncontrol@siemens.com
// stored: AutoNumber true, IsIECCheckEnabled false, IsRetainMemResEnabled false, MemoryReserve 100, SetENOAutomatically false, UDAEnableTagReadback false
   VAR
      instEventMgr_Alarm { ExternalAccessible := 'False'; ExternalVisible := 'False'; ExternalWritable := 'False'; S7_SetPoint := 'True'} : "CPG_EventManager";   // instance FB - Event Manager - Alarm Events
      instEventMgr_Warning { ExternalAccessible := 'False'; ExternalVisible := 'False'; ExternalWritable := 'False'; S7_SetPoint := 'True'} : "CPG_EventManager";   // instance FB - Event Manager - Warning Events
      instEventMgr_Status { ExternalAccessible := 'False'; ExternalVisible := 'False'; ExternalWritable := 'False'; S7_SetPoint := 'True'} : "CPG_EventManager";   // instance FB - Event Manager - Status Events
      instStatus_AlarmNotReset { ExternalAccessible := 'False'; ExternalVisible := 'False'; ExternalWritable := 'False'; S7_SetPoint := 'True'} : "CPG_Event";   // instance FB - PackML Event - Alarms not reset
      statEventMgr_Cmd_Reset { ExternalAccessible := 'False'; ExternalVisible := 'False'; ExternalWritable := 'False'} : Bool;   // Reset Cmd for all event managers
      statEventMgr_Cmd_Clear1stFlt { ExternalAccessible := 'False'; ExternalVisible := 'False'; ExternalWritable := 'False'} : Bool;   // Clear 1st Fault Cmd for all event managers
      statEventMgr_Clear1stFlt_OS { ExternalAccessible := 'False'; ExternalVisible := 'False'; ExternalWritable := 'False'} : Bool;   // Clear 1st Fault Cmd - One shot
   END_VAR
   VAR_TEMP   // added for the SCL form of the ladder/FBD networks
      _w1 : Bool;
      _w2 : Bool;
   END_VAR
BEGIN

REGION Network 1: ** STATE MODEL REPORTING STATUS ****
END_REGION

REGION Network 2: *** Call the PackML Module Initialize Logic ***
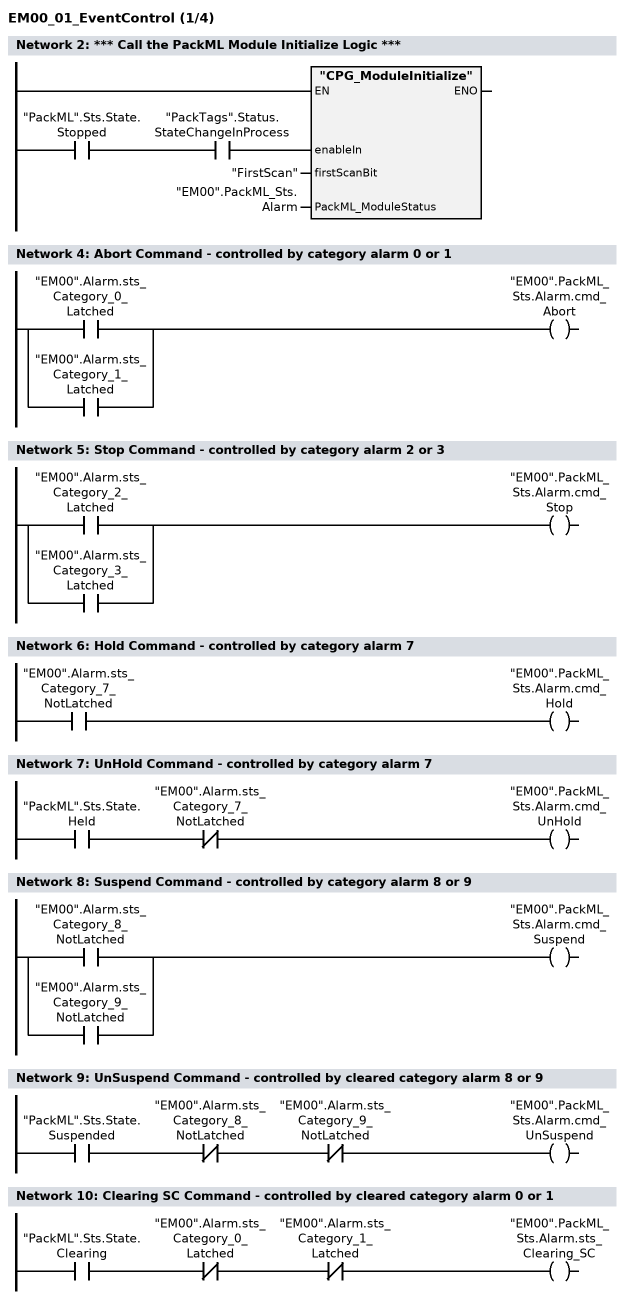
   RUNG wire#powerrail
      "CPG_ModuleInitialize"(enableIn := wire#w1, firstScanBit := "FirstScan", PackML_ModuleStatus := "EM00".PackML_Sts.Alarm)
   END_RUNG
   RUNG wire#powerrail
      Contact( "PackML".Sts.State.Stopped )
      Contact( "PackTags".Status.StateChangeInProcess )
   END_RUNG wire#w1
   // the same network as SCL:
   "CPG_ModuleInitialize"(enableIn := "PackML".Sts.State.Stopped AND "PackTags".Status.StateChangeInProcess,
                          firstScanBit := "FirstScan",
                          PackML_ModuleStatus := "EM00".PackML_Sts.Alarm);
END_REGION

REGION Network 3: Begin the LOGIC section.
END_REGION

REGION Network 4: Abort Command - controlled by category alarm 0 or 1
   RUNG wire#powerrail
      Contact( "EM00".Alarm.sts_Category_0_Latched )
      wire#w1
      Coil( "EM00".PackML_Sts.Alarm.cmd_Abort )
   END_RUNG
   RUNG wire#powerrail
      Contact( "EM00".Alarm.sts_Category_1_Latched )
   END_RUNG wire#w1
   // the same network as SCL:
   "EM00".PackML_Sts.Alarm.cmd_Abort := "EM00".Alarm.sts_Category_0_Latched OR "EM00".Alarm.sts_Category_1_Latched;
END_REGION

REGION Network 5: Stop Command - controlled by category alarm 2 or 3
   RUNG wire#powerrail
      Contact( "EM00".Alarm.sts_Category_2_Latched )
      wire#w1
      Coil( "EM00".PackML_Sts.Alarm.cmd_Stop )
   END_RUNG
   RUNG wire#powerrail
      Contact( "EM00".Alarm.sts_Category_3_Latched )
   END_RUNG wire#w1
   // the same network as SCL:
   "EM00".PackML_Sts.Alarm.cmd_Stop := "EM00".Alarm.sts_Category_2_Latched OR "EM00".Alarm.sts_Category_3_Latched;
END_REGION

REGION Network 6: Hold Command - controlled by category alarm 7
   RUNG wire#powerrail
      Contact( "EM00".Alarm.sts_Category_7_NotLatched )
      Coil( "EM00".PackML_Sts.Alarm.cmd_Hold )
   END_RUNG
   // the same network as SCL:
   "EM00".PackML_Sts.Alarm.cmd_Hold := "EM00".Alarm.sts_Category_7_NotLatched;
END_REGION

REGION Network 7: UnHold Command - controlled by category alarm 7
   RUNG wire#powerrail
      Contact( "PackML".Sts.State.Held )
      I_Contact( "EM00".Alarm.sts_Category_7_NotLatched )
      Coil( "EM00".PackML_Sts.Alarm.cmd_UnHold )
   END_RUNG
   // the same network as SCL:
   "EM00".PackML_Sts.Alarm.cmd_UnHold := "PackML".Sts.State.Held AND NOT "EM00".Alarm.sts_Category_7_NotLatched;
END_REGION

REGION Network 8: Suspend Command - controlled by category alarm 8 or 9
   RUNG wire#powerrail
      Contact( "EM00".Alarm.sts_Category_8_NotLatched )
      wire#w1
      Coil( "EM00".PackML_Sts.Alarm.cmd_Suspend )
   END_RUNG
   RUNG wire#powerrail
      Contact( "EM00".Alarm.sts_Category_9_NotLatched )
   END_RUNG wire#w1
   // the same network as SCL:
   "EM00".PackML_Sts.Alarm.cmd_Suspend := "EM00".Alarm.sts_Category_8_NotLatched OR "EM00".Alarm.sts_Category_9_NotLatched;
END_REGION

REGION Network 9: UnSuspend Command - controlled by cleared category alarm 8 or 9
   RUNG wire#powerrail
      Contact( "PackML".Sts.State.Suspended )
      I_Contact( "EM00".Alarm.sts_Category_8_NotLatched )
      I_Contact( "EM00".Alarm.sts_Category_9_NotLatched )
      Coil( "EM00".PackML_Sts.Alarm.cmd_UnSuspend )
   END_RUNG
   // the same network as SCL:
   "EM00".PackML_Sts.Alarm.cmd_UnSuspend := "PackML".Sts.State.Suspended AND NOT "EM00".Alarm.sts_Category_8_NotLatched AND NOT "EM00".Alarm.sts_Category_9_NotLatched;
END_REGION

REGION Network 10: Clearing SC Command - controlled by cleared category alarm 0 or 1
   RUNG wire#powerrail
      Contact( "PackML".Sts.State.Clearing )
      I_Contact( "EM00".Alarm.sts_Category_0_Latched )
      I_Contact( "EM00".Alarm.sts_Category_1_Latched )
      Coil( "EM00".PackML_Sts.Alarm.sts_Clearing_SC )
   END_RUNG
   // the same network as SCL:
   "EM00".PackML_Sts.Alarm.sts_Clearing_SC := "PackML".Sts.State.Clearing AND NOT "EM00".Alarm.sts_Category_0_Latched AND NOT "EM00".Alarm.sts_Category_1_Latched;
END_REGION

REGION Network 11: Resetting SC Command - controlled by cleared category alarm 0-3
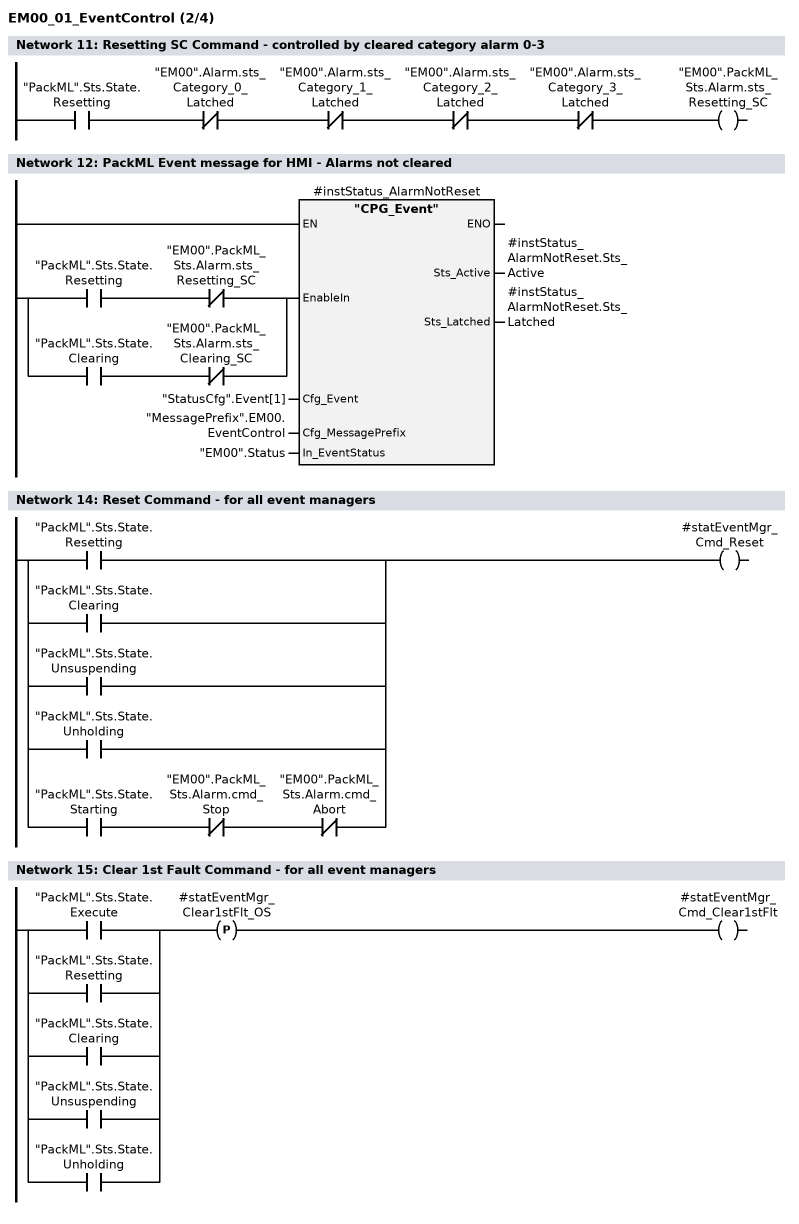
   RUNG wire#powerrail
      Contact( "PackML".Sts.State.Resetting )
      I_Contact( "EM00".Alarm.sts_Category_0_Latched )
      I_Contact( "EM00".Alarm.sts_Category_1_Latched )
      I_Contact( "EM00".Alarm.sts_Category_2_Latched )
      I_Contact( "EM00".Alarm.sts_Category_3_Latched )
      Coil( "EM00".PackML_Sts.Alarm.sts_Resetting_SC )
   END_RUNG
   // the same network as SCL:
   "EM00".PackML_Sts.Alarm.sts_Resetting_SC := "PackML".Sts.State.Resetting AND NOT "EM00".Alarm.sts_Category_0_Latched AND NOT "EM00".Alarm.sts_Category_1_Latched AND NOT "EM00".Alarm.sts_Category_2_Latched AND NOT "EM00".Alarm.sts_Category_3_Latched;
END_REGION

REGION Network 12: PackML Event message for HMI - Alarms not cleared
   RUNG wire#powerrail
      #instStatus_AlarmNotReset(EnableIn := wire#w1, Cfg_Event := "StatusCfg".Event[1], Cfg_MessagePrefix := "MessagePrefix".EM00.EventControl, In_EventStatus := "EM00".Status, Sts_Active => #instStatus_AlarmNotReset.Sts_Active, Sts_Latched => #instStatus_AlarmNotReset.Sts_Latched)
   END_RUNG
   RUNG wire#powerrail
      Contact( "PackML".Sts.State.Resetting )
      I_Contact( "EM00".PackML_Sts.Alarm.sts_Resetting_SC )
   END_RUNG wire#w1
   RUNG wire#powerrail
      Contact( "PackML".Sts.State.Clearing )
      I_Contact( "EM00".PackML_Sts.Alarm.sts_Clearing_SC )
   END_RUNG wire#w1
   // the same network as SCL:
   #instStatus_AlarmNotReset(EnableIn := ("PackML".Sts.State.Resetting AND NOT "EM00".PackML_Sts.Alarm.sts_Resetting_SC) OR ("PackML".Sts.State.Clearing AND NOT "EM00".PackML_Sts.Alarm.sts_Clearing_SC),   // "CPG_Event"
                           Cfg_Event := "StatusCfg".Event[1],
                           Cfg_MessagePrefix := "MessagePrefix".EM00.EventControl,
                           In_EventStatus := "EM00".Status,
                           Sts_Active => #instStatus_AlarmNotReset.Sts_Active,
                           Sts_Latched => #instStatus_AlarmNotReset.Sts_Latched);
END_REGION

REGION Network 13: *** EVENT CONTROL MANAGERS ***
END_REGION

REGION Network 14: Reset Command - for all event managers
   RUNG wire#powerrail
      Contact( "PackML".Sts.State.Resetting )
      wire#w1
      Coil( #statEventMgr_Cmd_Reset )
   END_RUNG
   RUNG wire#powerrail
      Contact( "PackML".Sts.State.Clearing )
   END_RUNG wire#w1
   RUNG wire#powerrail
      Contact( "PackML".Sts.State.Unsuspending )
   END_RUNG wire#w1
   RUNG wire#powerrail
      Contact( "PackML".Sts.State.Unholding )
   END_RUNG wire#w1
   RUNG wire#powerrail
      Contact( "PackML".Sts.State.Starting )
      I_Contact( "EM00".PackML_Sts.Alarm.cmd_Stop )
      I_Contact( "EM00".PackML_Sts.Alarm.cmd_Abort )
   END_RUNG wire#w1
   // the same network as SCL:
   #statEventMgr_Cmd_Reset := "PackML".Sts.State.Resetting OR "PackML".Sts.State.Clearing OR "PackML".Sts.State.Unsuspending OR "PackML".Sts.State.Unholding OR ("PackML".Sts.State.Starting AND NOT "EM00".PackML_Sts.Alarm.cmd_Stop AND NOT "EM00".PackML_Sts.Alarm.cmd_Abort);
END_REGION

REGION Network 15: Clear 1st Fault Command - for all event managers
   RUNG wire#powerrail
      Contact( "PackML".Sts.State.Execute )
      wire#w1
      P_Trig( #statEventMgr_Clear1stFlt_OS )
      Coil( #statEventMgr_Cmd_Clear1stFlt )
   END_RUNG
   RUNG wire#powerrail
      Contact( "PackML".Sts.State.Resetting )
   END_RUNG wire#w1
   RUNG wire#powerrail
      Contact( "PackML".Sts.State.Clearing )
   END_RUNG wire#w1
   RUNG wire#powerrail
      Contact( "PackML".Sts.State.Unsuspending )
   END_RUNG wire#w1
   RUNG wire#powerrail
      Contact( "PackML".Sts.State.Unholding )
   END_RUNG wire#w1
   // the same network as SCL:
   #_w1 := "PackML".Sts.State.Execute OR "PackML".Sts.State.Resetting OR "PackML".Sts.State.Clearing OR "PackML".Sts.State.Unsuspending OR "PackML".Sts.State.Unholding;
   #_w2 := #_w1 AND NOT #statEventMgr_Clear1stFlt_OS;   // rising edge
   #statEventMgr_Clear1stFlt_OS := #_w1;
   #statEventMgr_Cmd_Clear1stFlt := #_w2;
END_REGION

